		eManualRecipe_SelectedVariableType			: E_XMLVariableType; (* refer to E_XMLVariableType *)
		sManualRecipe_DefaultFilePath				: STRING := 'C:\SW\XML management\Recipe Handling';
		sManualRecipe_FileExtension					: STRING := 'XML';
(**)	sManualRecipe_sErrorMessage					: STRING;
(**)	iManualRecipe_TotalTimePv_100ms				: INT;
(**)	iManualRecipe_ExportedImportedQty			: INT;
(**)	iManualRecipe_ProgressPercentage			: INT;	

(**)	eManualRecipe_ImportExportMode				: E_XmlRWMode; (* refer to E_XmlRwMode :

														eXmlMode_MergeAllByType 					:= 1,			// SSER -> One XML, SSUR -> One XML, Product Recipe -> One XML and so on
														eXmlMode_SeperateByProductAndStation		:= 2,			// SSER will seperate by Station with Multiple file, same goes to the rest of the Recipe
														eXmlMode_SeperateAll					 	:= 3			// Seperate each of the recipe individually *)


	
	eHmiLanguage								: E_HmiLanguage;

	sHmiActiveUsername							: STRING(30):= 'TF2000 HMI User'; 	// Active username that login in HMI currently
	sHmiActiveUsergroup							: STRING(30);
	iHmiCurrentUserIDs							: INT := 1; 						// Standby for HMI Current User used
	ARsHmiUsernameList 							: ARRAY [0..50] OF STRING;			// HMI User Management Namelist push out from HMI
	ARsHmiUsergroupList 						: ARRAY [0..10] OF STRING;			// HMI User Management Namelist push out from HMI
	
	
	bEventRstPB									: BOOL; // Used in program, HMI and any places. This variable need to Mapped with Physical Input via FunctionBlock (FB3_EventModule)
	bBuzzerRstPB								: BOOL; // Used in program, HMI and any places. This variable need to Mapped with Physical Input via FunctionBlock (FB3_EventModule)
	bAcknowledgePB								: BOOL; // Used in program, HMI and any places. This variable need to Mapped with Physical Input via FunctionBlock (FB3_EventModule)
	


// Machine


	bShutdownRequestFlag						: BOOL;
	bManualRecipe_ReadyToShutdownFlag			: BOOL; // 
	bCSVWrite_ReadyToShutdownFlag				: BOOL; // 
	
	
// Boot Up Shut Down
	bMainCtrl									: BOOL;	
	bReadXmlEn									: BOOL;
	bReadXmlComplete							: BOOL;
	bMachineShutdown							: BOOL;
	bShutdownPopupPage							: BOOL;
	bRecipeShutdownRequestFlag					: BOOL;
	bCsvShutdownRequestFlag						: BOOL;
	bWriteXmlEn									: BOOL;
	bWrite_Done									: BOOL;
	bRead_Done									: BOOL;
	
	
// CSV Report Log
		
	dsCsvReport									: DS_CsvReport; // Please consider to change the naming of DS and declaration on upcoming project
	fbBkMemRingBuffer							: FB_MemRingBuffer;
	fbCsvHandler	 							: FB3_CsvHandler;
	sCsvFilePath								: STRING := 'C:\\report_csv\';
	udiCsvMRBCount								: UDINT;	// The number of data set stored in MRB (MemoryRingBuffer)
	udiCsvMRBUsagePercent 						: UDINT;	// Current Usage % in MRB (MemoryRingBuffer)
	ARdsCsvErrorLog								: ARRAY [1..C_iCsvErrorLogQty] OF DS_CsvErrorLog;
	dsCsvErrorLog_Empty							: DS_CsvErrorLog;

// CSV Event Log

	sCsvFilePath_EventLog						: STRING := 'C:\SW\EventLog\';

	
	
END_VAR
	
VAR_GLOBAL PERSISTENT
// Station, Loading, Unloading

//	ARiLdModulePickStnID						: ARRAY [0..C_iLdModuleQty] OF INT;  //XML_AutoRO_ManualRW  	// To "Name" the Loading Station with a Number, usually we will label the 1st Module Loading Conveyor with 79 (7=Loading, 9= the 9th Zone (or we all it max) of the conveyor end zone. 
//	ARiUldModuleUnloadStnID						: ARRAY [0..C_iUldModuleQty] OF INT; //XML_AutoRO_ManualRW		// To "Name" the Unlaoding Station with a Number, usually we will label the 1st Module of Unloading Conveyor with 81 (8=Unloading, 1=The 1st Zone of the unloading Conveyor.
	
// XML Multiple GVL Backup Version

	AR2sXMLMultipleGVLVerDate 				: ARRAY [1..C_iXMLSrvMultiGVLQty] OF ARRAY [1..C_iXMLMultipleGVLVerQty] OF STRING;

(***** CHECK ******


(* xxxxxxxxxxxxxxxxxxxxxxxxxxxxxxx  UPS - Internal Used xxxxxxxxxxxxxxxxxxxxxxxxxxxxxxx*)
(*========================================================================*)

	bGetUpsStatusEn						: BOOL := TRUE;
	bGetUpsStatusValid					: BOOL;
	bGetUpsStatusError					: BOOL;
	udiGetUpsStatusErrID					: UDINT;
	UpsStatus							: ST_UPSStatus;

(* xxxxxxxxxxxxxxxxxxxxxxxxxxxxxxx  UPS - External Used xxxxxxxxxxxxxxxxxxxxxxxxxxxxxxx*)
(*========================================================================*)
	(* --- Alarm --- *)
	bDCPowerUnknownStatusAlarm			: BOOL;
	bBatteryUnknownStatusAlarm			: BOOL;
	bUpsCommUnknownStatusAlarm		: BOOL;
	bBatteryReplacementRequestAlarm		: BOOL;
	bUpsCommErrorAlarm					: BOOL;
	(* --- Status --- *)
	bDCPowerModeActivated				: BOOL;
	bBatteryModeActivated				: BOOL;
	bUpsCommOkFlag					: BOOL;

	timeNow: TIMESTRUCT;

*)
	
(*
	// Arm
	C_iArmModuleQty 				: INT := 1; 								(* Total quantity of Single Arm + Multiple Arm Module - ex: 1x Multiple Arm (with 5 Vertical Axis) + 2x Single Arm = 3 Modules = Value: 3 *)
	C_ARiArmModuleVertAxisQty		: ARRAY [1..C_iArmModuleQty]OF INT := [1];	(* Total quantity of Veritical Axis per Arm Module *)
	C_ARMcArmHookQty				: INT := 1;									(* Total quantity of Hook per Machine, ex: 2x Arm Module, 1st Module with 1x Hook, 2nd Module is Multiple arm with 7x Hook, so thev value is add together = value: 8 *)

	// Station , Loading, Unloading	
	C_iProcessStnQty 						: INT := 6;		(* To change the Qty of Array*)
	C_iLdModuleQty					: INT := 1;		(* To Define Loading Group Set - How many module of Loading Conveyor*)
	C_iUldModuleQty					: INT := 1;		(* To Define Unloading Group Set - How many module of Unloading Conveyor*)
		
	C_ARiCvLdModuleZoneQty			: ARRAY [1..C_iLdStnQty] OF INT := [3];		(* Number of Zone on each of the Loading Conveyor Module (Module seperated by Array) *)
	C_ARiCvUldModuleZoneQty			: ARRAY [1..C_iUldStnQty] OF INT := [3];	(* Number of Zone on each of the Unloading Conveyor Module (Module seperated by Array) *)

	C_iTotalCvLdZoneQty				: INT := 3;		(* Number of Zone on each of the Loading Conveyor Module*)
	C_iTotalCvUldZoneQty			: INT := 3;		(* Number of Zone (Or Max Number of Zone) on each of the Unloading Conveyor Module*)
	*)

	
END_VAR

// ---- GVLs/GVL3/LIB_GVL_IO.TcGVL
{attribute 'Tc2GvlVarNames'}
VAR_GLOBAL


// Digital Input

	ARbDI						: ARRAY [0..C_iDigitalInputQty] OF BOOL;
	ARwMapDI					: ARRAY [100..C_iDigitalInputMappingChannelMaxID] OF WORD;
	ARwActualMapDI	AT %I* 		: ARRAY [1..10] OF WORD;

	
// Digital Output
	ARbDO						: ARRAY [0..C_iDigitalOutputQty] OF BOOL;
	ARwDO						: ARRAY [0..C_iDigitalOutputQty] OF WORD;
	ARwMapDO	 				: ARRAY [100..C_iDigitalOutputMappingChannelMaxID] OF WORD;
	ARwActualMapDO	AT %Q* 		: ARRAY [1..8] OF WORD;
	
// Deactivated

	ARbDeactivated				: ARRAY [0..C_iDigitalOutputQty] OF BOOL;

END_VAR

//VAR_GLOBAL CONSTANT

//	C_iDigitalInputQty					: INT := 220;		// Total Number of Digital Input Points
//	C_iDigitalOutputQty					: INT := 220;		// Total Number of Digital Output Points

//	C_iDigitalInputMappingChannelMaxID	: INT := 150;	// Max Channel ID of Digital Input Channel for Mapping Used (Ex: WX100 ~ WX116 ---> Value: 116
//	C_iDigitalOutputMappingChannelMaxID	: INT := 140; 	// Max Channel ID of Digital Output Channel for Mapping Used (Ex: WY100 ~ WY113 ---> Value: 113
	
//END_VAR

// ---- GVLs/GVL3/LIB_GVL_MEMORY.TcGVL
{attribute 'Tc2GvlVarNames'}
VAR_GLOBAL PERSISTENT
//	AR2dsSSMR						: ARRAY [0..C_iProcessStnQty] OF ARRAY [0..C_iSSMRRecipeQty] OF DS_SSMR;	//XML_AutoRW_ManualRW
//	AR2dsSSUR						: ARRAY [0..C_iProcessStnQty] OF ARRAY [0..C_iSSURRecipeQty] OF DS_SSUR;	//XML_AutoRW_ManualRW
//	AR2dsSSER 						: ARRAY [0..C_iProcessStnQty] OF ARRAY [0..C_iSSERRecipeQty] OF DS_SSER;	//XML_AutoRW_ManualRW
//	ARdsProductRecipe 				: ARRAY [0..C_iProRepRecipeQty] OF DS_ProductRecipe;						//XML_AutoRW_ManualRW

//	dsMcCarrierInfo					: DS_MachineCarrierInfo; 	// Previously call as BasketInfo
//	dsCarrierInfo_Empty				: DS_CarrierInfo;			// Empty DS
	
//	dsSSMR_Empty					: DS_SSMR;
//	dsSSUR_Empty					: DS_SSUR;
//	dsSSER_Empty					: DS_SSER;
//	dsProductRecipe_Empty			: DS_ProductRecipe;
	

	
END_VAR

// ---- GVLs/HMI_Ctrl/Global_Variables_CT12_HMIfunction.TcGVL
{attribute 'Tc2GvlVarNames'}
VAR_GLOBAL

	(*bAutoPageOn:BOOL;
	bManuPageOn:BOOL;
	bRecipePageOn: BOOL;	(*  *)
	bUserPageOn:BOOL;*)


	bSSURstartCOnditionPageOn:BOOL;


	(*bManualStationOnPage:BOOL;*)
	bAutoStationOnPage:BOOL;




END_VAR

// ---- GVLs/HMI_Ctrl/Global_Variables_HMI.TcGVL
{attribute 'Tc2GvlVarNames'}
VAR_GLOBAL

(*Simulator Screen*)

	bSimulatorPagePopUpFlag 							: BOOL;
	bAutoRecipeCallPage 									: BOOL;

	iRecipeSelectNo										: INT;

	bAutoRecipeBarcodeCallPage 							: BOOL;
	bBarcodePagePopUpFlag 								: BOOL;
	bAutoRecipeBarcodeClosePage 						: BOOL;

	sUserName											: STRING;



(*Yoges's Backup and Restore Apps*)

	restore : BOOL;
	backup : BOOL;
	otherwise : BOOL;
	dont : BOOL;
	ask : BOOL;
	me : BOOL;
	silent_backup : BOOL;


	iScrollbar : INT;

END_VAR

// ---- GVLs/HMI_Ctrl/Global_Variables_HMI_Function.TcGVL
{attribute 'Tc2GvlVarNames'}
VAR_GLOBAL PERSISTENT
(*Recipe Setting Page*)

	iStepNo:INT; (*RecipeEditorStepNoAssign*)
	iStationNo:INT;(*BasicRecipeStationNoAssign*)
	iArmStnNo :INT;(*ARm Setting Page*)
	iUsonicID:INT;(*UsonicIDno*)
	iUsonicID2:INT;
	sUltrasonicLabel:STRING;(*UsonicLabel/Name*)
	sUltrasonicLabel2 : STRING;
	iAutoInfoNo:INT;(*AutoMode Station Info Page No*)
	iManuPageNo:INT;(*Manul mode PAge No*)
	iArmControlPageNo:INT; (*Arm Page Control No*)
	OnOffStatus:INT; (*1=System Auto On, 2=System Auto Off*)
	lrVertHmiRatio:LREAL;(*ArmGraphicRatioMovement*)
	lrHorzHmiRatio:LREAL;(*ArmGraphicRatioMovement*)
	bFreqBtmChange: ARRAY [1..iStnQty] OF BOOL;
	bFreqSideChange: ARRAY [1..iStnQty] OF BOOL;	


	(*7day Auto On/Off(array1-On,2=off*)

	Day1En:ARRAY [1..2] OF BOOL;
	Day2En:ARRAY [1..2] OF BOOL;
	Day3En: ARRAY [1..2] OF BOOL;
	Day4En:ARRAY [1..2] OF BOOL;
	Day5En:ARRAY [1..2] OF BOOL;
	Day6En: ARRAY [1..2] OF BOOL;
	Day7En: ARRAY [1..2] OF BOOL;

	Day1H:ARRAY [1..2] OF INT;
	Day2H:ARRAY [1..2] OF INT;
	Day3H: ARRAY [1..2] OF INT;
	Day4H:ARRAY [1..2] OF INT;
	Day5H:ARRAY [1..2] OF INT;
	Day6H: ARRAY [1..2] OF INT;
	Day7H: ARRAY [1..2] OF INT;

	Day1M:ARRAY [1..2] OF INT;
	Day2M:ARRAY [1..2] OF INT;
	Day3M: ARRAY [1..2] OF INT;
	Day4M:ARRAY [1..2] OF INT;
	Day5M:ARRAY [1..2] OF INT;
	Day6M: ARRAY [1..2] OF INT;
	Day7M: ARRAY [1..2] OF INT;

	(*Arm Horizontal Position Remap*)
	Arm1HookPos: ARRAY [0..20] OF LREAL;
	Arm1UnHookPos: ARRAY [0..20] OF LREAL;

	Arm2HookPos: ARRAY [0..20] OF LREAL;
	Arm2UnHookPos: ARRAY [0..20] OF LREAL;

	bAutoPageOn:BOOL;
	bManuPageOn:BOOL;
	bRecipePageOn: BOOL;	(*  *)
	bUserPageOn:BOOL;
	bJRS_PageOn:BOOL;
	bGeneral_PageOn:BOOL;
         bDetergentMonitorAPageOn:BOOL;
         bDetergentMonitorBPageOn:BOOL;
         bVacuumMonitorPageOn:BOOL;
	bManualCalibratePageOn:BOOL;

	xRatio:LREAL;
	yRatio:LREAL;
	xRatio_1:LREAL;
	yRatio_1:LREAL;

	Arm1TopPos: ARRAY [0..iAddMapArrayLreal] OF LREAL;
	Arm1Pos1stStage: ARRAY [0..iAddMapArrayLreal] OF LREAL;
	Arm1Pos2ndStage: ARRAY [0..iAddMapArrayLreal] OF LREAL;
	Arm1Pos3rdStage: ARRAY [0..iAddMapArrayLreal] OF LREAL;
	Arm1Pos4thStage: ARRAY [0..iAddMapArrayLreal] OF LREAL;
	Arm1BottomPos: ARRAY [0..iAddMapArrayLreal] OF LREAL;
	Arm1MidPos: ARRAY [0..iAddMapArrayLreal] OF LREAL;

	Arm2TopPos: ARRAY [0..iAddMapArrayLreal] OF LREAL;
	Arm2Pos1stStage: ARRAY [0..iAddMapArrayLreal] OF LREAL;
	Arm2Pos2ndStage: ARRAY [0..iAddMapArrayLreal] OF LREAL;
	Arm2Pos3rdStage: ARRAY [0..iAddMapArrayLreal] OF LREAL;
	Arm2Pos4thStage: ARRAY [0..iAddMapArrayLreal] OF LREAL;
	Arm2BottomPos: ARRAY [0..iAddMapArrayLreal] OF LREAL;
	Arm2MidPos: ARRAY [0..iAddMapArrayLreal] OF LREAL;

END_VAR

VAR_GLOBAL

	iArmVertCurrentPos:INT;
	iArmHorzCurrentPos:INT;

	bArmPosSetPage:BOOL;
	bArm2PosSetPage : BOOL;


	bDeactivatePageOn:BOOL; (*Sensor Deactivated*)
	bStatusPreparationPageOn:BOOL;

	bArmJog2PageOn: BOOL;

	RecipeEditOn:BOOL; (*RecipeEditorEditPageCallUp*)

	bXML_ImportExportPageOn : BOOL;


	bStatusPreparePageOn:BOOL; (*Open Prepare Status Page*)
	bStatusOriginPageOn:BOOL;	(*Open Origin Status Page*)
	(*bAutoModeOtherDeactPageOn:BOOL;(*Open Deact. Others Page*)*)

	(*Time Tracker & Time Optimize Page*)

	TrackeriArrayNo: ARRAY [1..20] OF INT; (*Assign for tracker Array NO*)
	TimeTrackerPage:INT; (*Assign for tracker Page No*)


	(*Remap Arm Position Function*-because loading/unloading not in array form*)

	(*Produt Description for Recipe Edit*)
	sRecipeDescriptionStep : ARRAY [1..20] OF STRING;

	(*Arm Homing Complete Indicator*)
	bArmVertHomingComplete:BOOL;
	bArmHorzHomingComplete:BOOL;
	bArmHomingComplete: ARRAY [1..iArmQty] OF BOOL;

	(*Page On bit*)

	bAlarmPageOn:BOOL;
	bRecipeSubMenuPageOn:BOOL;

	(*Auto Mode Recipe Select*)
	bAutoModeRecipeSelect:BOOL;

	JogSlowPullOn:BOOL;
	JogArmOn:BOOL;

	(*Station On page bit*)
	bStationOnPage:BOOL;
	bManualStationOnPage:BOOL;
	bManualStationOffPage:BOOL;

	(*Manual Mode U/Sonic Power Set*)

	iUsonicA_PowerManuSV : ARRAY [1..20] OF INT;
	iUsonicB_PowerManuSV : ARRAY [1..20] OF INT;


	(*Detergent Basket Quatity (PV) Reset PB user password control*)
	ARiManualDetergentResetPassword 	: ARRAY [0..iStnQty] OF STRING;
	ARbManualDetergentResetFlag			: ARRAY [0..iStnQty] OF BOOL;

	bInputListOn:BOOL;
	bOutputListOn:BOOL;
	bRecipeListOn:BOOL;


	Xmove:INT;
	Ymove:INT;

	bStationOffPage: BOOL;
	RecipeEditOff:BOOL;
END_VAR

VAR_GLOBAL


END_VAR

// ---- GVLs/Internal Address/GVL_Internal_Variable.TcGVL
{attribute 'Tc2GvlVarNames'}
VAR_GLOBAL
	
	ARbMAP_ArmMisshookSensorA 				: ARRAY [1..iArmQty] OF BOOL;
	ARbMAP_ArmMisshookSensorB 				: ARRAY [1..iArmQty] OF BOOL;
	
	bMAP_LdConfirmBasketPickAvailibility	: BOOL;

END_VAR

// ---- GVLs/Memory_Ctrl/Global_Variables_Memory.TcGVL
{attribute 'Tc2GvlVarNames'}
VAR_GLOBAL PERSISTENT

(* xxxxxxxxxxxsxxxxxx BasketMemory - Basket Cfm/ Trf Internal Used xxxxxxxxsxxxxxxxxx*)
(*========================================================================*)

	fbLdBasketMemory					: ARRAY [0..iCvLdQty] OF fbV2_SingleArmBasketMemoryV2;
	fbA1StationBasketMemory				: ARRAY [0..iStnQty] OF fbV2_SingleArmBasketMemoryV2;
	fbA2StationBasketMemory				: ARRAY [0..iStnQty] OF fbV2_SingleArmBasketMemoryV2;
	fbUldBasketMemory					: ARRAY [0..iCvUldQty] OF fbV2_SingleArmBasketMemoryV2;

(* xxxxxxxxxxxxxxxxxxxxxxxxxxxx  BasketInfo - Internal Used xxxxxxxxxxxxxxxxxxxxxxxxxxxx*)
(*========================================================================*)

	DSLdBasketInfoConfirm 				: ARRAY [0..iLdStnQty] OF DSV2_BasketInfo;
	DSLdBasketInfoTransfer 				: ARRAY [0..iLdStnQty] OF DSV2_BasketInfo;

	DSUldBasketInfoConfirm 				: ARRAY [0..iUldStnQty] OF DSV2_BasketInfo;
	DSUldBasketInfoTransfer 				: ARRAY [0..iUldStnQty] OF DSV2_BasketInfo;

	DSStnBasketInfo						: ARRAY [0..iStnQty] OF DSV2_BasketInfo;
	DSArmBasketInfo 						: ARRAY [0..iArmQty] OF DSV2_BasketInfo;

(* xxxxxxxxxxxxxxxxxxxxx  BasketInfo - Loading / Unloading Conveyor Used xxxxxxxxxxxxxxxxxxxxx *)
(*================================================================================*)

	AR2sDSCv_LdConfirmBasketInfo 		: ARRAY [1..iLdStnQty, 1..iCvLdQty] OF DSV2_BasketInfo;
	AR2sDSCv_LdTransferBasketInfo 		: ARRAY [1..iLdStnQty, 1..iCvLdQty] OF DSV2_BasketInfo;

	AR2sDSCv_UldConfirmBasketInfo 		: ARRAY [1..iUldStnQty, 1..iCvUldQty] OF DSV2_BasketInfo;
	AR2sDSCv_UldTransferBasketInfo 		: ARRAY [1..iUldStnQty, 1..iCvUldQty] OF DSV2_BasketInfo;

(* xxxxxxxxxxxxxxxxxxxxx  Station Memory and InputOutput Variable - Internal Used xxxxxxxxxxxxxxxxxxxxx*)
(*=====================================================================================*)

	LdDSStationSSERStore				: DSV2_fbStationSequenceRecipeStore;
	LdDSStationSSURStore 				: DS_fbStationSubRecipeStore;

	LdDSStationSSERCall					: DSV2_fbStationSequenceRecipeCall;
	LdDSStationSSURCall 					: DS_fbStationSubRecipeCall;

	ARDsStnSeqProInput 					: ARRAY [0..iStnQty] OF DS_StnSeqProInput;
	ARDSStnSeqProOutput 				: ARRAY [0..iStnQty] OF DS_StnSeqProOutput;

	AR10DSStationSSERStore				: ARRAY [0..iStnQty] OF DSV2_fbStationSequenceRecipeStore;
	AR10DSStationSSERCall				: ARRAY [0..iStnQty] OF DSV2_fbStationSequenceRecipeCall;

	AR10DSStationSSURStore 				: ARRAY [0..iStnQty] OF DS_fbStationSubRecipeStore;
	AR10DSStationSSURCall 				: ARRAY [0..iStnQty] OF DS_fbStationSubRecipeCall;

(* xxxxxxxxxxxxxxxxxxxxxxxxxxxxx  Station Process Variable - Internal Used xxxxxxxxxxxxxxxxxxxxxxxxxxxxx*)
(*=====================================================================================*)

	fbMainStationProcess_Stn				: ARRAY [1..iStnQty] OF fbV2_MainStationProcess;
	ARDsStnSeqProcessCtrl 				: ARRAY [0..iStnQty] OF DS_fbStnSeqProcessCtrl;
	ARbProductRecipeCallEn 				: ARRAY [0..iStnQty] OF BOOL;
	ARiProductRecipeNoCall 				: ARRAY [0..iStnQty] OF INT;
	ARiProductRecipeStepCall 				: ARRAY [0..iStnQty] OF INT;
	DSfbGnrProductRecipeMemoryOut 		: DSV2_fbGnrProductRecipeMemoryOut;
	ARiStnNoToCalledArm					: ARRAY [0..iArmQty] OF INT;
	ARDSGnrFeedArmPnpParameter		: ARRAY [0..iArmQty] OF DSV2_Gnr_CalledArmPnpParameter;
	ARbArmReady						: ARRAY [1..iArmQty] OF BOOL;								(* Universal*) (* Input  - From ArmPnpFB, This signal is used to confirm if the arm is ready and idling*)
	ARbStationProcessCompletedFlag		: ARRAY [0..iStnQty] OF BOOL;

(*xxxxxxxxxxxxxxxxxxxxxxxxxxx fbGnrProductRecipeMemory - Internal Used xxxxxxxxxxxxxxxxxxxxxxxxxxx*)
(*=====================================================================================*)

(*Input/Output*)
	ARiCurrentHorzStnNo					: ARRAY [1..iArmQty] OF INT;
	ARi1StepPatternNo					: ARRAY [1..iArmQty] OF INT;
	ARDs1StepUpDownMovement			: ARRAY [1..iArmQty] OF DSA1_UpDownMovement;
	ARi4StepPatternNo					: ARRAY [1..iArmQty] OF INT;
	ARDs4StepUpDownMovement			: ARRAY [1..iArmQty] OF DSA1_UpDownMovement;

(* xxxxxxxxxxxxxxxxxxxxxxxxxxx  Station ZoneHeight Variable - External Used xxxxxxxxxxxxxxxxxxxxxxxxxxx*)
(*=====================================================================================*)

	ARDSLdZoneHeight 					: ARRAY [0..iLdStnQty] OF DSA32_StationZoneHeight;
	ARDSStationZoneHeight 				: ARRAY [0..iStnQty] OF DSA32_StationZoneHeight;
	ARDSUldZoneHeight 					: ARRAY [0..iUldStnQty] OF DSA32_StationZoneHeight;

(* xxxxxxxxxxxxxxxxxxxxxxxxxxx  Station ZoneHeight Variable - Internal Used xxxxxxxxxxxxxxxxxxxxxxxxxxx*)
(*=====================================================================================*)

	ARDSLdZonePosOut					: ARRAY [0..iLdStnQty] OF DSA32_StationZonePosOut; (*From fbGnrProductRecipeMemory Output*)
	ARDSStationZonePosOut 				: ARRAY [0..iStnQty] OF DSA32_StationZonePosOut; (*From fbGnrProductRecipeMemory Output*)
	ARDSUldZonePosOut 					: ARRAY [0..iUldStnQty] OF DSA32_StationZonePosOut;(*From fbGnrProductRecipeMemory Output*)

(* xxxxxxxxxxxxxxxxxxxxxxxxxxxxx  MaxMin Time Used  xxxxxxxxxxxxxxxxxxxxxxxxxxxxx*)
(*====================================================================*)

	ARDsSSERSourceMinMaxTime_Uni		: ARRAY [1..iStnQty] OF DSV2_SSERSourceMinMaxTime;
	ARDsStnMinMaxEffTimeDisplay			: ARRAY [0..iStnQty] OF DSV2_StnMinMaxEffTIme;
	DSV2MTBMinMaxEffTime 				: DSV2_MinMaxEffTime;

(* xxxxxxxxxxxxxxxxxxxxx  IndusoftScreenMapping - External Used xxxxxxxxxxxxxxxxxxxxx*)
(*========================================================================*)

	DSScrMapSSUR 						: DS_fbStationSubRecipeStore;
	DSScrMapSSER 						: DSV2_fbStationSequenceRecipeStore;
	iCurrentScreenNo						: INT;

(* xxxxxxxxxxxxxxxxxxxxx  Indusoft Product Recipe Description Display control  -  xxxxxxxxxxxxxxxxxxxxxxxxxx*)

	ARsUpPickPatternDescription			: ARRAY [0..iProductRecipeStepArrayQty] OF STRING(50);
	ARsDownTransferPatternDescription		: ARRAY [0..iProductRecipeStepArrayQty] OF STRING(50);

(*Indusoft*)
	sProductRecipeStep1SeqRecipeDescription: STRING(50);
	sProductRecipeStep2SeqRecipeDescription: STRING(50);
	sProductRecipeStep3SeqRecipeDescription: STRING(50);
	sProductRecipeStep4SeqRecipeDescription: STRING(50);
	sProductRecipeStep5SeqRecipeDescription: STRING(50);
	sProductRecipeStep6SeqRecipeDescription: STRING(50);
	sProductRecipeStep7SeqRecipeDescription: STRING(50);
	sProductRecipeStep8SeqRecipeDescription: STRING(50);
	sProductRecipeStep9SeqRecipeDescription: STRING(50);
	sProductRecipeStep10SeqRecipeDescription: STRING(50);
	sProductRecipeStep11SeqRecipeDescription: STRING(50);
	sProductRecipeStep12SeqRecipeDescription: STRING(50);
	sProductRecipeStep13SeqRecipeDescription: STRING(50);
	sProductRecipeStep14SeqRecipeDescription: STRING(50);
	sProductRecipeStep15SeqRecipeDescription: STRING(50);
	sProductRecipeStep16SeqRecipeDescription: STRING(50);
	sProductRecipeStep17SeqRecipeDescription: STRING(50);
	sProductRecipeStep18SeqRecipeDescription: STRING(50);
	sProductRecipeStep19SeqRecipeDescription: STRING(50);
	sProductRecipeStep20SeqRecipeDescription: STRING(50);

	ARsUpPickPatternDescription1: STRING(50);
	ARsUpPickPatternDescription2: STRING(50);
	ARsUpPickPatternDescription3: STRING(50);
	ARsUpPickPatternDescription4: STRING(50);
	ARsUpPickPatternDescription5: STRING(50);
	ARsUpPickPatternDescription6: STRING(50);
	ARsUpPickPatternDescription7: STRING(50);
	ARsUpPickPatternDescription8: STRING(50);
	ARsUpPickPatternDescription9: STRING(50);
	ARsUpPickPatternDescription10: STRING(50);
	ARsUpPickPatternDescription11: STRING(50);
	ARsUpPickPatternDescription12: STRING(50);
	ARsUpPickPatternDescription13: STRING(50);
	ARsUpPickPatternDescription14: STRING(50);
	ARsUpPickPatternDescription15: STRING(50);
	ARsUpPickPatternDescription16: STRING(50);
	ARsUpPickPatternDescription17: STRING(50);
	ARsUpPickPatternDescription18: STRING(50);
	ARsUpPickPatternDescription19: STRING(50);
	ARsUpPickPatternDescription20: STRING(50);

	ARsDownTransferPatternDescription1: STRING(50);
	ARsDownTransferPatternDescription2: STRING(50);
	ARsDownTransferPatternDescription3: STRING(50);
	ARsDownTransferPatternDescription4: STRING(50);
	ARsDownTransferPatternDescription5: STRING(50);
	ARsDownTransferPatternDescription6: STRING(50);
	ARsDownTransferPatternDescription7: STRING(50);
	ARsDownTransferPatternDescription8: STRING(50);
	ARsDownTransferPatternDescription9: STRING(50);
	ARsDownTransferPatternDescription10: STRING(50);
	ARsDownTransferPatternDescription11: STRING(50);
	ARsDownTransferPatternDescription12: STRING(50);
	ARsDownTransferPatternDescription13: STRING(50);
	ARsDownTransferPatternDescription14: STRING(50);
	ARsDownTransferPatternDescription15: STRING(50);
	ARsDownTransferPatternDescription16: STRING(50);
	ARsDownTransferPatternDescription17: STRING(50);
	ARsDownTransferPatternDescription18: STRING(50);
	ARsDownTransferPatternDescription19: STRING(50);
	ARsDownTransferPatternDescription20: STRING(50);

END_VAR

// ---- GVLs/ModbusTCP_Ctrl/Global_Variables_Modbus.TcGVL
{attribute 'Tc2GvlVarNames'}
VAR_GLOBAL

(******** Modbus TCP variable declaration - as a SLAVE ********)  (*** If as a MASTER, then don't need to declare this variable***)

   	mb_Input_Coils        		: ARRAY [0..255] OF BOOL;
    	mb_Output_Coils      	 	: ARRAY [0..255] OF BOOL;
    	mb_Input_Registers    		: ARRAY [0..255] OF WORD;
    	mb_Output_Registers   		: ARRAY [0..255] OF WORD;

	bOutputRegisterAddr0		: BOOL;

END_VAR

// ---- GVLs/Others TBD/Globale_VarCheck.TcGVL
{attribute 'Tc2GvlVarNames'}
VAR_GLOBAL
	CheckBounds_ErrCnt:INT;
	CheckByteZeroDiv_ErrCnt:INT;
	CheckDintZeroDiv_ErrCnt:INT;
	CheckDWordZeroDiv_ErrCnt:INT;
	CheckIntZeroDiv_ErrCnt:INT;
	CheckLrealZeroDiv_ErrCnt:INT;
	CheckRealZeroDiv_ErrCnt:INT;
	CheckSIntZeroDiv_ErrCnt:INT;
	CheckWordZeroDiv_ErrCnt:INT;
	CheckRangeSigned_ErrCnt:INT;
	CheckRangeUnsigned:INT;
END_VAR

// ---- GVLs/Others TBD/Global_HMI.TcGVL
{attribute 'Tc2GvlVarNames'}
VAR_GLOBAL

	bAutoModeOnPB		:BOOL;
	bAutoPrepareStatus		:BOOL;
	bBarcodeRegisterPageON	:BOOL;
	bManualModeOnPB	:BOOL;
	bRecipeModeOnPB	:BOOL;
	bRecipeSSUROnPB		:BOOL;
	bRecipeSSEROnPB		:BOOL;
	bRecipeBasicOnPB		:BOOL;
	bRecipeBasic2OnPB		:BOOL;
	bRecipeProductOnPB		:BOOL;
	bRecipeOtherOnPB		:BOOL;
	bRecipeTimeOptimizeOnPB:BOOL;
	bRecipeArmSettingOnPB	:BOOL;
	bRecipeArmSetting2OnPB	:BOOL;
	bAlarmModeOnPB	:BOOL;
	bUserModeOnPB		:BOOL;

	bManualCalibrate		:BOOL;
	bAutoModeOperationStatusPage:	BOOL;


	bAutoModeOn	:BOOL;
	bManualModeOn	:BOOL;
	bRecipeModeOn	:BOOL;
	bRecipeSSUROn	:BOOL;
	bRecipeSSEROn	:BOOL;
	bRecipeBasicOn	:BOOL;
	bRecipeBasic2On	:BOOL;
	bRecipeProductOn:BOOL;
	bRecipeOtherOn	:BOOL;
	bRecipeTimeOptimizeOn:BOOL;
	bRecipeArmSettingOn	:BOOL;
	bRecipeArmSetting2On:BOOL;
	bAlarmModeOn	:BOOL;
	bUserModeOn	:BOOL;
	bSchematicPageOn :BOOL;

	bManualModeOnLatch :BOOL;	(*to call Confirm Pop Up page Manual Out*)
	bManualOutToAutoConfirmPageOn	:BOOL; (*Manual Out Pop Up Page to Auto On bit*)
	bManualOutToRecipeConfirmPageOn	:BOOL; (*Manual Out Pop Up Page to Recipe On bit*)
	bManualOutToUserConfirmPageOn	:BOOL; (*Manual Out Pop Up Page to User On bit*)
	bManualOutLatchCfm				:BOOL; (*Use as a latch bit for timer to reset All Page bit On PB*)
	
	bManualModeOffLatch :BOOL;	(*to exit Confirm Pop Up page Manual Out*)
	bManualOutToAutoConfirmPageOff	:BOOL; (*Manual Out Pop Up Page to Auto Off bit*)
	bManualOutToRecipeConfirmPageOff	:BOOL; (*Manual Out Pop Up Page to Recipe Off bit*)
	bManualOutToUserConfirmPageOff	:BOOL; (*Manual Out Pop Up Page to User Of bit*)




	(*iStationNo		:INT;*)



	bAutoModeOnRE		:R_TRIG;
	bManualModeOnRE	:R_TRIG;
	bRecipeModeOnRE	:R_TRIG;
	bRecipeSSUROnRE	:R_TRIG;
	bRecipeBasicOnRE	:R_TRIG;
	bRecipeBasic2OnRE	:R_TRIG;
	bRecipeSSEROnRE	:R_TRIG;
	bRecipeProductOnRE   :R_TRIG;
	bRecipeOtherOnRE	:R_TRIG;
	bRecipeTimeOptimizeOnRE:R_TRIG;
	bRecipeArmSettingOnRE	:R_TRIG;
	bRecipeArmSetting2OnRE	:R_TRIG;
	bAlarmModeOnRE	:R_TRIG;
	bUserModeOnRE		:R_TRIG;

	bLoadingPageSeqCompleteRE	:R_TRIG;
	bManualModeOnLatchFE	:F_TRIG;


(*Initial Loading Page Timer*)

	bAutoModeOnTON	:TON;
	bManualModeOnTON	:TON;
	bRecipeModeOnTON	:TON;
	bRecipeSSUROnTON	:TON;
	bRecipeSSEROnTON	:TON;
	bRecipeBasicOnTON	:TON;
	bRecipeBasic2OnTON	:TON;
	bRecipeProductOnTON:TON;
	bRecipeOtherOnTON	:TON;
	bRecipeTimeOptimizeOnTON:TON;
	bRecipeArmSettingOnTON	:TON;
	bRecipeArmSetting2OnTON :TON;
	bAlarmModeOnTON	:TON;
	bUserModeOnTON	:TON;
	bManualOutLatchCfmTON 	:TON;


	bAutoModeOnSeq	:BOOL;
	bManualModeOnSeq	:BOOL;
	bRecipeModeOnSeq	:BOOL;
	bRecipeSSUROnSeq	:BOOL;
	bRecipeSSEROnSeq	:BOOL;
	bAlarmModeOnSeq	:BOOL;
	bUserModeOnSeq	:BOOL;
         bRecipeBasicOnSeq	:BOOL;
         bRecipeBasic2OnSeq	:BOOL;
         bRecipeProductOnSeq		:BOOL;
	bRecipeOtherOnSeq		:BOOL;
	bRecipeTimeOptimizeOnSeq:BOOL;
	bRecipeArmSettingOnSeq	:BOOL;
	bRecipeArmSetting2OnSeq	:BOOL;


(*Password Save Confirm page*)
	bSaveCfmPB: BOOL;
	bSaveCfmPageOn: BOOL;
	bSaveBufferPB:BOOL;
	bSavePageCnfmOnRE: R_TRIG;
	sUserPasswordSave: STRING;
	tBackupDelayOffTimer: TON;
	bIncorrectPswdOn: BOOL;
	bSaveBufferPBRE: R_TRIG;



(*Xml Execute Push Button*)
	bExecuteWriteXml		: BOOL;
	bExecuteReadXml	:BOOL;
	bErrorReadXml		:BOOL;


(*Secs\Gem Command Page Call*)

	bSecGemsPageON 									:BOOL;

(*Recipe Selection Mode*)

	sRecipeSelectionStatus								:STRING;

(*SECS\GEM Selection Mode Message*)

	sSecGemSelectionButtonMessage						:STRING;

	sRemotCommandStateMessage						:STRING;





	bLoadingPageSeqComplete	:BOOL;
	
	ARdsMAP_HmiVariableStn		: ARRAY[1..iStnQty] OF DS_HMI_MappingVariable;
	ARdsMAP_HmiVariableGeneral	: DS_HMI_MappingVariable;

	
END_VAR

// ---- GVLs/Others TBD/Global_Variables_Lib_NonPresistent.TcGVL
{attribute 'Tc2GvlVarNames'}
VAR_GLOBAL

(*Global Variable for FunctionBlock in Library *)

	(* HMI Declaration *)
	iHMIRecipeNo				: INT;
	bRecipeLoadPb				: BOOL;
	bRecipeSavePb				: BOOL;
	bProductRecipeClearPb		: BOOL;
	bClearPB_SSER 				: ARRAY [1..6] OF BOOL;
	bClearPB_SSUR 				: ARRAY [1..6] OF BOOL;
	bClearPB_SSER_Uni			: BOOL;
	bClearPB_SSUR_Uni			: BOOL;
	

	(*XML Handler & XML Fb*)
	iXMLRecipeNo				: INT := 1;
	FBXmlSrvRead				:  FB_XmlSrvRead;
	FBXmlSrvWrite				:  FB_XmlSrvWrite;
	DSV3XML_Recipe			: DSV3_XML_Recipe;

	ARiSubAction					: ARRAY [1..10] OF INT; (* 0-Idle, 1-Import, 2-Export, 3-Clear/Delete 8-Done *)



	(*SecsGem Simulation Used Only*)

	iSecsGemRecipeNo			: INT := 1;

	iSecsGemLoadHS			: INT; 				(* S7F1/S7F2 		: 0-Idle, 1-Enable, 2-Busy, 3-Done, 4-Error *)
	iSecsGemSentHS				: INT; 				(* S7F3/S7F4 		: 0-Idle, 1-Enable, 2-Busy, 3-Done, 4-Error *)
	iSecsGemRequestHS			: INT; 				(* S7F5/S7F6 		: 0-Idle, 1-Enable, 2-Busy, 3-Done, 4-Error *)
	iSecsGemDeleteHS			: INT; 				(* S7F17/S7F18 	: 0-Idle, 1-Enable, 2-Busy, 3-Done, 4-Error *)


	(* Declared for S7F18 -> Delete Request *)
	ARDsPnpSequenceMemory_Delete 									: ARRAY [1..iProductRecipeArrayQty] OF DSV2_A1_PnpSequenceMemory;
	AR3SiRecipeTimeBlockMemoryNoCallArmTime_Delete				    : ARRAY [1..iProductRecipeArrayQty, 1..iRecipeBlockQty, 1..9] OF INT;
	AR3SiRecipeTimeBlockMemoryWithCallArmTime_Delete				: ARRAY [1..iProductRecipeArrayQty, 1..iRecipeBlockQty, 1..9] OF INT;
	ARbProductRecipeTimeBlockAvailable_Delete 						: ARRAY [0..iProductRecipeArrayQty] OF BOOL;
	ARDSTempCtrlRecipe_Delete 										: ARRAY [0..iProductRecipeArrayQty] OF DSV3_TempCtrlRecipe;


END_VAR

// ---- GVLs/Others TBD/Global_Variables_Lib_Persistent.TcGVL
{attribute 'Tc2GvlVarNames'}
VAR_GLOBAL PERSISTENT


	ARiLdStnID								: ARRAY [1..iLdStnQty] OF INT;		(* To Define Loading Station ID*)
	ARiUldStnID								: ARRAY [1..iUldStnQty] OF INT;		(* To Define Unloading Station ID*)

	ARDSTempCtrlRecipe 					: ARRAY [0..iProductRecipeArrayQty] OF DSV3_TempCtrlRecipe;  (* Used by fbV3_TemperatureParaRecipe, Make it Global so that future can read/write easily*)

END_VAR

// ---- GVLs/Others TBD/Global_Variables_PID.TcGVL
{attribute 'Tc2GvlVarNames'}
VAR_GLOBAL

	No_input							: INT;
	Ratio								: INT;
	InvRatio							: INT;

	Stn1FlowRawData				: INT;
	Stn2FlowRawData				: INT;
	Stn3FlowRawData				: INT;
	Stn4FlowRawData				: INT;
	Stn5FlowRawData				: INT;
	Stn6FlowRawData				: INT;
	Stn7FlowRawData				: INT;
	ARiStnFlowRawData				: ARRAY [1..iStnQty] OF INT;

	Stn1ActualFlowRawData		: INT;
	Stn2ActualFlowRawData		: INT;
	Stn3ActualFlowRawData		: INT;
	Stn4ActualFlowRawData		: INT;
	Stn5ActualFlowRawData		: INT;
	Stn6ActualFlowRawData		: INT;
	Stn7ActualFlowRawData		: INT;
	ARiStnActualFlowRawData	: ARRAY [1..iStnQty] OF INT;


	Stn1U_SonicOn				: BOOL;
	Stn2U_SonicOn				: BOOL;
	Stn3U_SonicOn				: BOOL;
	Stn4U_SonicOn				: BOOL;
	Stn5U_SonicOn				: BOOL;
	Stn6U_SonicOn				: BOOL;
	Stn7U_SonicOn				: BOOL;
	ARiStnU_SonicOn			: ARRAY [1..iStnQty] OF BOOL;

	Pump1_Freq_Reading			: REAL;
	Pump2_Freq_Reading			: REAL;
	Pump3_Freq_Reading			: REAL;
	Pump4_Freq_Reading			: REAL;
	Pump5_Freq_Reading			: REAL;
	Pump6_Freq_Reading			: REAL;
	Pump7_Freq_Reading			: REAL;

	Pump1_Freq_Actual			: INT;
	Pump2_Freq_Actual			: INT;
	Pump3_Freq_Actual			: INT;
	Pump4_Freq_Actual			: INT;
	Pump5_Freq_Actual			: INT;
	Pump6_Freq_Actual			: INT;
	Pump7_Freq_Actual			: INT;

	Pump1_Freq_Reading_Raw	: INT;
	Pump2_Freq_Reading_Raw	: INT;
	Pump3_Freq_Reading_Raw	: INT;
	Pump4_Freq_Reading_Raw	: INT;
	Pump5_Freq_Reading_Raw	: INT;
	Pump6_Freq_Reading_Raw	: INT;
	Pump7_Freq_Reading_Raw	: INT;

	Stn1Actual_LPM				: INT;
	Stn2Actual_LPM				: INT;
	Stn3Actual_LPM				: INT;
	Stn4Actual_LPM				: INT;
	Stn5Actual_LPM				: INT;
	Stn6Actual_LPM				: INT;
	Stn7Actual_LPM				: INT;

	Pump1FlowAlarm				: BOOL;
	Pump2FlowAlarm				: BOOL;
	Pump3FlowAlarm				: BOOL;
	Pump4FlowAlarm				: BOOL;
	Pump5FlowAlarm				: BOOL;
	Pump6FlowAlarm				: BOOL;
	Pump7FlowAlarm				: BOOL;
	
	//Heater
	Stn8TempRawData				: INT;
	Stn9TempRawData				: INT;
	Stn10TempRawData			: INT;



END_VAR

// ---- GVLs/Others TBD/Global_Variables_PID_1.TcGVL
{attribute 'Tc2GvlVarNames'}
VAR_GLOBAL PERSISTENT


	Stn1PumpHiFlowSV		:INT;
	Stn2PumpHiFlowSV		:INT;
	Stn3PumpHiFlowSV		:INT;
	Stn4PumpHiFlowSV		:INT;
	Stn5PumpHiFlowSV		:INT;
	Stn6PumpHiFlowSV		:INT;
	Stn7PumpHiFlowSV		:INT;
	ARiStnPumpHiFlowSV	:ARRAY [1..iStnQty] OF INT;


	Stn1PumpLowFlowSV	:INT;
	Stn2PumpLowFlowSV	:INT;
	Stn3PumpLowFlowSV	:INT;
	Stn4PumpLowFlowSV	:INT;
	Stn5PumpLowFlowSV	:INT;
	Stn6PumpLowFlowSV	:INT;
	Stn7PumpLowFlowSV	:INT;
	ARiStnPumpLowFlowSV	: ARRAY [1..iStnQty] OF INT;

	ARiStnManualPumpLowFlowSV :ARRAY [1..iStnQty] OF INT;
	ARiStnManualPumpHighFlowSV :ARRAY [1..iStnQty] OF INT;


END_VAR

// ---- GVLs/Others TBD/GVL_HMI_CKK.TcGVL
{attribute 'Tc2GvlVarNames'}
VAR_GLOBAL


	
	iBufferPage											: INT;
	iSelectedPage										: INT;
	iReturnPage											: INT;
	bManualPageOn										: BOOL;
	bManualExitConfirm									: BOOL;
	bManualExitCancel									: BOOL;
	bBlockBasketEnter									: BOOL;
iCkkTest	: DINT;


iDisplayTimeCycle : ARRAY [1..iStnQty] OF REAL; 
bDisplayTimeCycleOn : ARRAY [1..iStnQty] OF BOOL;
iDisplayTimeCycleEnd : ARRAY [1..iStnQty] OF INT;
ARiStnProcessTimeCD : ARRAY [1..iStnQty] OF INT;
ARsStnProcessName : ARRAY [1..iStnQty] OF STRING;
iAutoStnInfoPageNo	: INT :=1;
ARsHMIDisplaySSURDescription	: ARRAY [1..IStationSubRecipeArrayQty] OF STRING;
iSettingStnNo	: INT :=1;
iSettingStnNoBuffer	: INT :=1;
iArmSettingStnNo : INT :=1;
iArmSettingStnNoBuffer : INT :=1;
sDisplayConductivity : ARRAY [1..2] OF STRING;
bDosingPageEn		 : ARRAY [1..iStnQty] OF BOOL;
iConfigSSER			 : ARRAY [1..20] OF INT;
bSelectTempExternal	 : ARRAY [1..4] OF BOOL;
bSelectTempExternalInd : ARRAY [1..4] OF BOOL;
iSelectTempExternal	 : INT;
bBarcodeRegPage		 : BOOL;
iDisplayFreqUs		 : ARRAY [1..iStnQty] OF INT;
iDisplayRecipeFreqUs : INT;

sBasketNo			 : STRING;
bBarcodeConfirm		 : BOOL;

bParameterPopupPageOn : BOOL;

bPopupPageRapidPBOn: BOOL;
bPopupPageRapidConfirm: BOOL;
bBarcodeCallPagePB		: BOOL;

// Barcode
sBarcodeScannerReceivedResult: STRING;
	iBarcodeRegUserSelectRecipeNo			: INT;
	iBarcodeRegUserSelectNoDataToSave		: INT;
	bBarcodeRegSave							: BOOL;
	bBarcodeRegClear						: BOOL;
	//bBarcodeEmpty							: BOOL;
	
	bBufferClearPB_SSER 				: ARRAY [1..6] OF BOOL;
	bBufferClearPB_SSUR 				: ARRAY [1..6] OF BOOL;
	
	tClearPB_SSER_Timer 				: ARRAY [1..6] OF TON;
	tClearPB_SSUR_Timer 				: ARRAY [1..6] OF TON;
	
	
END_VAR

// ---- GVLs/PDF_Report/Global_Variables_PDF_Report.TcGVL
{attribute 'Tc2GvlVarNames'}
VAR_GLOBAL

	sNameUser	:STRING;													(*Map with User login Name*)

	a1_dataLink								: ARRAY [1..100] OF ST_DataLog;
	a2_dataLink								: ARRAY [1..100] OF ST_DataLog;
	a3_dataLink								: ARRAY [1..100] OF ST_DataLog;
	a4_dataLink								: ARRAY [1..100] OF ST_DataLog;
	a5_dataLink								: ARRAY [1..100] OF ST_DataLog;
	a6_dataLink								: ARRAY [1..100] OF ST_DataLog;
	a7_dataLink								: ARRAY [1..100] OF ST_DataLog;
	a8_dataLink								: ARRAY [1..100] OF ST_DataLog;
	a9_dataLink								: ARRAY [1..100] OF ST_DataLog;
	a10_dataLink								: ARRAY [1..100] OF ST_DataLog;
	a11_dataLink								: ARRAY [1..100] OF ST_DataLog;
	a12_dataLink								: ARRAY [1..100] OF ST_DataLog;

	sLdtittle								: STRING;
	sStn1tittle								: STRING;
	sStn2tittle								: STRING;
	sStn3tittle								: STRING;
	sStn4tittle								: STRING;
	sStn5tittle								: STRING;
	sStn6tittle								: STRING;
	sStn7tittle								: STRING;
	sStn8tittle								: STRING;
	sStn9tittle								: STRING;
	sStn10tittle								: STRING;
	sStn11tittle								: STRING;
	sStn12tittle								: STRING;
	sStn13tittle								: STRING;

	
	ARsLdBasketInTime 					: ARRAY [0..iLdStnQty] OF STRING;
	ARsStnBasketInTime 					: ARRAY [0..iStnQty] OF STRING;
	ARsStnBasketOutTime 				: ARRAY [0..iStnQty] OF STRING;
	ARsUldBasketInTime 					: ARRAY [0..iUldStnQty] OF STRING;
	
	ARiLdBasketProductRecipeBuffer 		: ARRAY [0..iLdStnQty] OF INT;
	ARsLdBasketNoBuffer 				: ARRAY [0..iLdStnQty] OF STRING;
	
	ARiStnBasketProductRecipeBuffer 	: ARRAY [0..iStnQty] OF INT;
	ARsStnBasketNoBuffer 				: ARRAY [0..iStnQty] OF STRING;
	
	ARiUldBasketProductRecipeBuffer 	: ARRAY [0..iUldStnQty] OF INT;
	ARsUldBasketNoBuffer 				: ARRAY [0..iUldStnQty] OF STRING;
	
END_VAR

VAR_GLOBAL PERSISTENT

	iProgBatchTotal							:INT; (*For Unique nobor for each file*)

END_VAR

// ---- GVLs/Process_Ctrl/Global_Variables_Process_NoPersistent.TcGVL
{attribute 'Tc2GvlVarNames'}
VAR_GLOBAL

(* xxxxxxxxxxxxxxxxxxxxxxx DosingPumpControl Process Variable xxxxxxxxxxxxxxxxxxxxxxx*)
(*========================================================================*)

(*Input*)
	ARbStnErrorReset										: ARRAY [1..iStnQty] OF BOOL;
	ARbStnDrainST										: ARRAY [1..iStnQty] OF BOOL;
	ARbStnManualDosingST 								: ARRAY [1..iStnQty] OF BOOL;
	ARbStnFirstFillST										: ARRAY [1..iStnQty] OF BOOL;
	ARbStnAutoDosingST									: ARRAY [1..iStnQty] OF BOOL;

(*Output*)

	ARbStnAutoDosingDone 								: ARRAY [1..iStnQty] OF BOOL;
	ARbStnManualDosingDone 							: ARRAY [1..iStnQty] OF BOOL;
	ARbStnFirstFillInProgress 								: ARRAY [1..iStnQty] OF BOOL;
	ARbStnAutoDosingInProgress 							: ARRAY [1..iStnQty] OF BOOL;
	ARbStnManualDosingInProgress 						: ARRAY [1..iStnQty] OF BOOL;
	ARbStnPumpHealthCheckPulseError						: ARRAY [1..iStnQty] OF BOOL;

	ARiStnHealthCheckPulsePV							: ARRAY [1..iStnQty] OF INT;

	ARbStnFirstFillingHR									: ARRAY [1..iStnQty] OF BOOL;
	ARbStnFirstFillDone									: ARRAY [1..iStnQty] OF BOOL;

(* xxxxxxxxxxxxxxxxxxxxxxxxxxxxx Conveyor Motor Control xxxxxxxxxxxxxxxxxxxxxxxxxxxxx*)
(*========================================================================*)

	ARbLdIndexPB 										: ARRAY [0..iLdStnQty] OF BOOL;
	ARsLdConvStatus										: ARRAY [0..iLdStnQty] OF STRING;

	ARbUldIndexPB 										: ARRAY [0..iUldStnQty] OF BOOL;
	ARsUldConvStatus									: ARRAY [0..iUldStnQty] OF STRING;

	ARbLdConveyorIdErrorFlag 							: ARRAY [1..iCvLdQty] OF BOOL;
	ARbUldConveyorIdErrorFlag 							: ARRAY [1..iCvUldQty] OF BOOL;

	ARtLdIndexPBDelayTimePV 							: ARRAY [0..iLdStnQty] OF TIME;
	ARtLdRapidPBDelayTimePV 							: ARRAY [0..iLdStnQty] OF TIME;
	ARtLdTimerBasedRapidDelayTimePV					: ARRAY [0..iLdStnQty] OF TIME;
	ARtLdIndexConfirmDelayTimePV 						: ARRAY [0..iLdStnQty] OF TIME;
	ARtLdEndZoneDelayTimePV 							: ARRAY [0..iLdStnQty] OF TIME;

	ARtUldIndexPBDelayTimePV 							: ARRAY [0..iUldStnQty] OF TIME;
	ARtUldRapidPBDelayTimePV 							: ARRAY [0..iUldStnQty] OF TIME;
	ARtUldTimerBasedRapidDelayTimePV					: ARRAY [0..iUldStnQty] OF TIME;
	ARtUldIndexConfirmDelayTimePV 						: ARRAY [0..iUldStnQty] OF TIME;
	ARtUldEndZoneDelayTimePV 							: ARRAY [0..iUldStnQty] OF TIME;

	bConveyorStartInternal									: BOOL;
	bConveyorInternal											: BOOL	;

	Ld1ConvFb											: fbV2_LdUldCvCtrl;
	Uld1ConvFb											: fbV2_LdUldCvCtrl;
	Uld2ConvFb											: fbV2_LdUldCvCtrl;

	fbV2LdCv5zonewith5m5sCtrl								: fbV2_Cv5zonewith5m5sCtrl;
	fbV2LdCv4zonewith4m4sCtrl								: fbV2_Cv4zonewith4m4sCtrl;
	fbV2LdCv3zonewith3m3sCtrl								: fbV2_Cv3zonewith3m3sCtrl;
	bLdCvBasketEndReached								: BOOL;
	bLdCvBasketFull										: BOOL;

	fbV2UldCv5zonewith5m5sCtrl							: fbV2_Cv5zonewith5m5sCtrl;
	fbV2UldCv4zonewith4m4sCtrl							: fbV2_Cv4zonewith4m4sCtrl;
	fbV2UldCv3zonewith3m3sCtrl							: fbV2_Cv3zonewith3m3sCtrl;
	bUldCvBasketEndReached								: BOOL;
	bUldCvBasketFull										: BOOL;

(* xxxxxxxxxxxxxxxxxxxxxxxxxxxxx AutoPreparation Variable xxxxxxxxxxxxxxxxxxxxxxxxxxxxx*)
(*========================================================================*)

	ARtStnDelayOffTopupTimerOn							: ARRAY [0..iStnQty] OF TON;
	ARtStnSubTankDelayOffTopupTimerOn					: ARRAY [0..iStnQty] OF TON;
	ARtMainTankDelayOffTopupTimerOn						: TON;
	ARtMainTankRowDelayOffTopupTimerOn					: TON;
	ARtLoadingRowDelayOffTopupTimerOn					: TON;

	ARtStnTimeEV										: ARRAY [0..iStnQty] OF TIME;
	ARtStnSubTankTimeEV								: ARRAY [0..iStnQty] OF TIME;
(* xxxxxxxxxxxxxxxxxxxxxxxxxx Manual Drain Process Variable xxxxxxxxxxxxxxxxxxxxxxxxxx*)
(*========================================================================*)

	ARtStnDrainLowLevelDelayTimer						: ARRAY [0..iStnQty] OF TON;

	ARtStnDrainDelayEV									: ARRAY [0..iStnQty] OF TIME;

	bManualAllTankDrainEn 								: BOOL;
	bManualAllTankDrainCompletedFlag						: BOOL;

(* xxxxxxxxxxxxxxxxxxxxxxxxxx  Process Variable xxxxxxxxxxxxxxxxxxxxxxxxxx*)
(*========================================================================*)

	ARbStnCylinderInOutCtrl 								: ARRAY [1..iStnQty] OF BOOL;
	ARbStnCylinderOriginFlag								: ARRAY [1..iStnQty] OF BOOL;

(* xxxxxxxxxxxxxxxxxxxxxxxxxxx Vacuum Drain Variable Cltr xxxxxxxxxxxxxxxxxxxxxxxxxxx*)
(*========================================================================*)

	bCCtankDrainDone									: BOOL;
	bManualClearWaterTrap								: BOOL;
	bStnManualDrainCut									: BOOL;

(* xxxxxxxxxxxxxxxxxxxxxxxxxxxxxxxx General Process Variable xxxxxxxxxxxxxxxxxxxxxxxxxxxxxxxx*)
(*========================================================================*)

	ARiStnToleranceTimePV								: ARRAY [0..iStnQty] OF INT;
	ARbStnAssignBadBskBit								: ARRAY [0..iStnQty] OF BOOL;
	bBasketMissingReset									: BOOL;


(* xxxxxxxxxxxxxxxxxxxxxxxxxxxxxxxx Station Min  Process Time Displayed Variable xxxxxxxxxxxxxxxxxxxxxxxxxxxxxxxx*)
(*========================================================================*)
	fbV3TotalProcessTimeTracker							: fbV3_TotalProcessTimeTracker;
	ARiStationMinTimeDisplay								: ARRAY [1..iStnQty] OF INT;
	sStationDescriptionDisplay								: STRING;



END_VAR

// ---- GVLs/Process_Ctrl/Global_Variables_Process_Persistent.TcGVL
{attribute 'Tc2GvlVarNames'}
VAR_GLOBAL PERSISTENT

(* xxxxxxxxxxxxxxxxxxxxxxx DosingPumpControl Process Variable xxxxxxxxxxxxxxxxxxxxxxx*)
(*========================================================================*)

	ARDSProminentDosingHMI 									: ARRAY [1..iStnQty] OF DS_ProminentDosingHMI;
	ARfbProminentDosingCtrl									: ARRAY [1..iStnQty] OF fbProminentDosingCtrl;

	ARiStnPulseOnTime_ms									: ARRAY [1..iStnQty] OF INT;
	ARiStnPulseOffTime_ms 									: ARRAY [1..iStnQty] OF INT;
	ARiStnPumpFeedbackPulseInputFilter_ms 					: ARRAY [1..iStnQty] OF INT;
	ARiStnPumpHealthCheckPulseSV 							: ARRAY [1..iStnQty] OF INT;

(* xxxxxxxxxxxxxxxxxxxxxxxxxxxxx Conveyor Motor Control xxxxxxxxxxxxxxxxxxxxxxxxxxxxx*)
(*========================================================================*)

	ARrLdIndexPBDelayTimeSV_Sec 							: ARRAY [0..iLdStnQty] OF REAL;
	ARrLdRapidPBDelayTimeSV_Sec 							: ARRAY [0..iLdStnQty] OF REAL;
	ARrLdIndexConfirmDelayTimeSV_Sec 						: ARRAY [0..iLdStnQty] OF REAL;
	ARrLdEndZoneDelayTimeSV_Sec 							: ARRAY [0..iLdStnQty] OF REAL;

	ARrUldIndexPBDelayTimeSV_Sec 							: ARRAY [0..iUldStnQty] OF REAL;
	ARrUldRapidPBDelayTimeSV_Sec 							: ARRAY [0..iUldStnQty] OF REAL;
	ARrUldIndexConfirmDelayTimeSV_Sec 						: ARRAY [0..iUldStnQty] OF REAL;
	ARrUldEndZoneDelayTimeSV_Sec 							: ARRAY [0..iUldStnQty] OF REAL;

	diUnloadingTimer										: DINT;
	diUnloadingSingleBasketReachedTimer						: DINT;
	diUnloadingBuzzerOffHeaterTimer							: DINT;
	iUldBasketDelayPushTimerSV_sec							: INT;
	iUldBasketDelayPushTimeCountDown						: INT;
	diLdReturnConvMotorDelayOffTimer						: DINT;
	diUldReturnConvMotorDelayOffTimer						: DINT;

	rLdConveyorPos1ConfirmDelayTimeSV_Sec 					: REAL;
	rLdConveyorPos2ConfirmDelayTimeSV_Sec 					: REAL;
	rLdConveyorPos3ConfirmDelayTimeSV_Sec 					: REAL;
	rLdConveyorPos4ConfirmDelayTimeSV_Sec 					: REAL;

	rLdConveyorPos1ConfirmDelayOnTimeSV_Sec 				: REAL;
	rLdConveyorPos2ConfirmDelayOnTimeSV_Sec 				: REAL;
	rLdConveyorPos3ConfirmDelayOnTimeSV_Sec 				: REAL;
	rLdConveyorPos4ConfirmDelayOnTimeSV_Sec 				: REAL;
	
	rUldConveyorPos1ConfirmDelayTimeSV_Sec 					: REAL;
	rUldConveyorPos2ConfirmDelayTimeSV_Sec 					: REAL;
	rUldConveyorPos3ConfirmDelayTimeSV_Sec 					: REAL;
	rUldConveyorPos4ConfirmDelayTimeSV_Sec 					: REAL;

	rUldConveyorPos1ConfirmDelayOnTimeSV_Sec 				: REAL;
	rUldConveyorPos2ConfirmDelayOnTimeSV_Sec 				: REAL;
	rUldConveyorPos3ConfirmDelayOnTimeSV_Sec 				: REAL;
	rUldConveyorPos4ConfirmDelayOnTimeSV_Sec 				: REAL;

(* xxxxxxxxxxxxxxxxxxxxxxxxxxx General Process Variable xxxxxxxxxxxxxxxxxxxxxxxxxxx*)
(*======================================================================*)

	ARiStnToleranceTimeSV									: ARRAY [0..iStnQty] OF INT;
	ARiArmToleranceTimeSV									: ARRAY [0..iArmQty] OF INT;

	ARbRecipeSelectedFlag									: ARRAY [1..iProductRecipeArrayQty] OF BOOL;

         ARbOptionSelectedAutoTopupFlag						          : ARRAY [1..iProductRecipeArrayQty] OF BOOL;
         ARbOptionSelectedRecipeFlag						      	  	 : ARRAY [1..iProductRecipeArrayQty] OF BOOL;

(* xxxxxxxxxxxxxxxxxxxxxxxxxxx Arm related in Process xxxxxxxxxxxxxxxxxxxxxxxxxxx*)
(*======================================================================*)

	tAllStnArmTake											: INT;
	ARiStnDippingTimeSV										: ARRAY [1..iStnQty] OF INT;
	iFFUDelayOffTimerSV_min									: INT;
	iStnAgitation1DelayOffTimerSV_min							: INT;
	iStnAgitation2DelayOffTimerSV_min							: INT;

(* xxxxxxxxxxxxxxxxxxxxxxxxxxxxx Valve related in Process  xxxxxxxxxxxxxxxxxxxxxxxxxxxxx*)

	iAllTankLowLevelDelayTimeSV 							: INT;
	ARiLoadingTopUpDelayOffTimeSV 							: INT;
	ARiStnTopUpDelayOffTimeSV								: ARRAY [1..iStnQty] OF INT;
	ARiStnSubTankTopUpDelayOffTimeSV						: ARRAY [1..iStnQty] OF INT;

	ARiStnTopUpMaxTimeCutOffSV								: ARRAY [1..iStnQty] OF INT;

	iVacuumDrainSV											: INT;

	bBasketPushBasedTimer									: BOOL;

	ARbIncomingDIValveBasedDetergent						: ARRAY [1..iStnQty] OF BOOL;

	iCylinderBasketBackDelayTimeSV							: INT;
	iCylinderBasketFrontDelayTimeSV							: INT;

	iStn3PumpHzSV												: INT;

(* xxxxxxxxxxxxxxxxxxxxxxxxxxxxxxxx Dryer Cooling Ctrl xxxxxxxxxxxxxxxxxxxxxxxxxxxxxxxx*)
(*========================================================================*)

	ARfbV2DryerCoolingCtrlStn 									: ARRAY [1..iStnQty] OF fbV2_DryerCoolingCtrl;
	ARsStnDryerCoolingStatus									: ARRAY [1..iStnQty] OF STRING;
	ARiStnHeaterOnTimeActivation_Sec 							: ARRAY [1..iStnQty] OF INT ;
	ARiStnBlowerDelayOffTime_min								: ARRAY [1..iStnQty] OF INT ;

END_VAR

// ---- GVLs/RecycleMachineJRSCtrl/Global_Variables_JRS_HMI.TcGVL
{attribute 'Tc2GvlVarNames'}
VAR_GLOBAL

(*JRS_HMI Function*)

	JrsHmiPage:INT;
	bChillerManualPageOn:BOOL;
	bChillerAutoPageOn:BOOL;
	bManulBoilPageOn:BOOL;


END_VAR

// ---- GVLs/RecycleMachineJRSCtrl/Global_Variables_RecycleJRS.TcGVL
{attribute 'Tc2GvlVarNames'}
VAR_GLOBAL PERSISTENT

	DSV3_JRSHMI 											: DSV3_JRS_HMI; (*Channel of Other Digitial IO and DT*)

END_VAR

VAR_GLOBAL

	fbV3JRSModuleWithChiller									: fb_V3JRSModuleWithChiller;

	DSV3_JRSAlarm 											: DSV3_JRS_Alarm; (*Channel 200 ~ 204*)
	DSV3_JRSInput 											: DSV3_JRS_Input; (*Channel 0 ~ 3 *)
	DSV3_JRSOutput 											: DSV3_JRS_Output; (*Channel 100 ~ 103*)


END_VAR

// ---- GVLs/Secs_Gem/Global_Secs_Gem.TcGVL
{attribute 'Tc2GvlVarNames'}
VAR_GLOBAL

(*Machine Status & Control*)
(*-----------------------------------------------------------------------------------------------------------------------------------------------------------------------------------------------------------------------------------------------------------------*)

	(*Remote Command*)
	iRemote_Command_State : INT; (*Command from Secs/Gem to remote machine (Function only in Online Remote)
								 0 - Idle, 1 - INIT, 2 - RESET, 3 - START, 4 - STOP, 5 - PP-SELECT*)

	(*(*Control State-In Persisten Page*)
	iSecs_Control_State :INT;	(* Determine in Gem Console. Machine react base on this setting
							3 - Offline (Secs/GEM Offline - Remote Command disable)
							4 - Online Local (Secs/GEM Online - Local Control - Remote Command disable)
							5 - Online Remote (Secs/Gem Online - Host Control - Remote Command enable)*)*)

	(*Machine Status/ Process Status*)
	iMachine_Status :INT; 		(*Update Secs/Gem the Machine Status
							1 - INIT, 2 - READY, 3 - RUNNING, 4 - ALARM, 5 - STOP*)

	iSecGemStationNo	:INT; (*To refresh the station no for data (Constant Variable*)
(*Control State*)



(*-----------------------------------------------------------------------------------------------------------------------------------------------------------------------------------------------------------------------------------------------------------------*)



(*Production Info /Basket Info*)
(*-----------------------------------------------------------------------------------------------------------------------------------------------------------------------------------------------------------------------------------------------------------------*)

	(*Input Basket ID*)
	(*AR2sDSCv_LdConfirmBasketInfo[1,1].sProgramDescription		:STRING; (*Update Secs/Gem the Basket In ID UPH - Secs/Gem able to capture the start process
																	  (Update Sequence - PPExecName -> Input Basket ID)*)
	(*Output Basket ID*)
	AR2sDSCv_UldConfirmBasketInfo[1,3].sProgramDescription		:STRING;  (*Update Secs/Gem the Basket Out ID, Result & Counter UPH - Secs/Gem able to capture the end process
																	   (Update Sequence - Output Basket Result -> Output Basket Counter -> Output Basket ID)*)
	(*Output Basket Result*)
	AR2sDSCv_UldConfirmBasketInfo[1,3].bAvailibility				:BOOL;

	(*Output Basket Counter*)*)
	(*diTotalBasketQty_Customer								:INT;*)


	bBasketQuality: BOOL;		(*Basket Quality identification- Good= True; Bad= False*)
(*Alarm*)
(*---------------------------------------------------------------------------------------------------------------------------------------------------------------------------------------------------------------------------------------------------------------------*)

(*ARbAlarmOutput-using global alarm*)

(*Recipe*)
(*----------------------------------------------------------------------------------------------------------------------------------------------------------------------------------------------------------------------------------------------------------------------------*)

	(*PPChangeStatus*)
	iSecsGemPPchange 		:INT;		(*Update Secs/Gem that PLC already create/Edit/Delete the recipe
											PPChangeStatus - Action done by PLC (0-Idle, 1-Created, 2-Edited, 3-Deleted)*)
	iSecsGemPPchangeName	:INT;			(*PPChangeName - Selected recipe*)

	(*PPExecName*)
	(*AR2sDSCv_LdConfirmBasketInfo[1,1].iProductRecipeNo*)         (*Update Secs/Gem the selected recipe to run the current basket*)

	(*PP-SelectName-server send Product No if the Remote Host is Enable/ON*)
	iServerSecsGemProgNo		:INT;


	(*HMI_Function.iRecipeNoFeed	-(Server Monitor), iServerSecsGemProgNo-(From server)  :INT;	(*During Online Remote Mode (PP-SELECT), Secs/Gem order machine to run this recipe*)*)

	(*PPDirectory*)
	sRecipeFileDirectory			:STRING(200);	(*Share folder for PLC to output all recipes. Collect the persistent data and configuration file from the Boot folder ?C:\TwinCAT\Boot*)

	(*PPUpdateStatus*)
	iSecsGemPPupdate		:INT;		(*Secs/Gem to inform PLC that specific recipe is already downloaded
										PPUpdateStatus - (0-Idle, 1-Created, 2-Edited, 3-Deleted)-once the file overwite is complete, SecsGem will write '2' to the Address. Use the same address (iSecsGemWriteCompleted)*)
	iSecsGemPPupdateName	:INT;		(*PPUpdateName - Selected recipe*)

	(*PPLog*)
	sSecsGemRecipeWriteLog		:ARRAY [0..4] OF STRING(200);	(*LabView will log 5 udated recipe event for PLC (to display at PLC)*)







END_VAR

// ---- GVLs/Secs_Gem/Global_Variables_Secs_Gem_Persistent.TcGVL
{attribute 'Tc2GvlVarNames'}
VAR_GLOBAL PERSISTENT


	iSecs_Control_State :INT;	(* Determine in Gem Console. Machine react base on this setting
							3 - Offline (Secs/GEM Offline - Remote Command disable)
							4 - Online Local (Secs/GEM Online - Local Control - Remote Command disable)
							5 - Online Remote (Secs/Gem Online - Host Control - Remote Command enable)*)

END_VAR

// ---- GVLs/SevenDay_Ctrl/Global_Variables_Process_Door.TcGVL
{attribute 'Tc2GvlVarNames'}
VAR_GLOBAL

(* xxxxxxxxxxxxxxxxxxxxxxxxxxxxxxxx Ld Door Variable xxxxxxxxxxxxxxxxxxxxxxxxxxxxxxxx*)
(*========================================================================*)

	wLdDoorOpen									: WORD;
	bLdDoorOpen_00									: BOOL;
	bLdDoorOpen_01									: BOOL;
	bLdDoorOpen_02									: BOOL;
	bLdDoorOpen_03									: BOOL;
	bLdDoorOpen_04									: BOOL;
	bLdDoorOpen_05									: BOOL;
	bLdDoorOpen_06									: BOOL;
	bLdDoorOpen_07									: BOOL;
	bLdDoorOpen_08									: BOOL;
	bLdDoorOpen_09									: BOOL;
	bLdDoorOpen_10									: BOOL;
	bLdDoorOpen_11									: BOOL;
	bLdDoorOpen_12									: BOOL;
	bLdDoorOpen_13									: BOOL;
	bLdDoorOpen_14									: BOOL;
	bLdDoorOpen_15									: BOOL;

	wLdDoorClose									: WORD;
	bLdDoorClose_00									: BOOL;
	bLdDoorClose_01									: BOOL;
	bLdDoorClose_02									: BOOL;
	bLdDoorClose_03									: BOOL;
	bLdDoorClose_04									: BOOL;
	bLdDoorClose_05									: BOOL;
	bLdDoorClose_06									: BOOL;
	bLdDoorClose_07									: BOOL;
	bLdDoorClose_08									: BOOL;
	bLdDoorClose_09									: BOOL;
	bLdDoorClose_10									: BOOL;
	bLdDoorClose_11									: BOOL;
	bLdDoorClose_12									: BOOL;
	bLdDoorClose_13									: BOOL;
	bLdDoorClose_14									: BOOL;
	bLdDoorClose_15									: BOOL;

	bLdDoorOpenCompleted							: BOOL;
	bLdDoorCloseCompleted							: BOOL;

	bLdDoorOpenAct									: BOOL;
	bLdDoorCloseAct									: BOOL;

(*HoldingBitSV*)

	bLdDoorOpenHolding								: BOOL;
	bLdDoorCloseHolding								: BOOL;
	bLdDoorClampHolding								: BOOL;
	bLdDoorUnClampHolding							: BOOL;

(* xxxxxxxxxxxxxxxxxxxxxxxxxxxxxxxx Stn1 Door Variable xxxxxxxxxxxxxxxxxxxxxxxxxxxxxxxx*)
(*========================================================================*)

	wStn1DoorOpen										: WORD;
	bStn1DoorOpen_00									: BOOL;
	bStn1DoorOpen_01									: BOOL;
	bStn1DoorOpen_02									: BOOL;
	bStn1DoorOpen_03									: BOOL;
	bStn1DoorOpen_04									: BOOL;
	bStn1DoorOpen_05									: BOOL;
	bStn1DoorOpen_06									: BOOL;
	bStn1DoorOpen_07									: BOOL;
	bStn1DoorOpen_08									: BOOL;
	bStn1DoorOpen_09									: BOOL;
	bStn1DoorOpen_10									: BOOL;
	bStn1DoorOpen_11									: BOOL;
	bStn1DoorOpen_12									: BOOL;
	bStn1DoorOpen_13									: BOOL;
	bStn1DoorOpen_14									: BOOL;
	bStn1DoorOpen_15									: BOOL;

	wStn1DoorClose										: WORD;
	bStn1DoorClose_00									: BOOL;
	bStn1DoorClose_01									: BOOL;
	bStn1DoorClose_02									: BOOL;
	bStn1DoorClose_03									: BOOL;
	bStn1DoorClose_04									: BOOL;
	bStn1DoorClose_05									: BOOL;
	bStn1DoorClose_06									: BOOL;
	bStn1DoorClose_07									: BOOL;
	bStn1DoorClose_08									: BOOL;
	bStn1DoorClose_09									: BOOL;
	bStn1DoorClose_10									: BOOL;
	bStn1DoorClose_11									: BOOL;
	bStn1DoorClose_12									: BOOL;
	bStn1DoorClose_13									: BOOL;
	bStn1DoorClose_14									: BOOL;
	bStn1DoorClose_15									: BOOL;

	bStn1DoorOpenCompleted								: BOOL;
	bStn1DoorCloseCompleted								: BOOL;

	bStn1DoorOpenAct									: BOOL;
	bStn1DoorCloseAct									: BOOL;

(*HoldingBitSV*)

	bStn1DoorOpenHolding								: BOOL;
	bStn1DoorCloseHolding								: BOOL;
	bStn1DoorClampHolding								: BOOL;
	bStn1DoorUnClampHolding								: BOOL;

(* xxxxxxxxxxxxxxxxxxxxxxxxxxxxxxxx Stn2 Door Variable xxxxxxxxxxxxxxxxxxxxxxxxxxxxxxxx*)
(*========================================================================*)

	wStn2DoorOpen										: WORD;
	bStn2DoorOpen_00									: BOOL;
	bStn2DoorOpen_01									: BOOL;
	bStn2DoorOpen_02									: BOOL;
	bStn2DoorOpen_03									: BOOL;
	bStn2DoorOpen_04									: BOOL;
	bStn2DoorOpen_05									: BOOL;
	bStn2DoorOpen_06									: BOOL;
	bStn2DoorOpen_07									: BOOL;
	bStn2DoorOpen_08									: BOOL;
	bStn2DoorOpen_09									: BOOL;
	bStn2DoorOpen_10									: BOOL;
	bStn2DoorOpen_11									: BOOL;
	bStn2DoorOpen_12									: BOOL;
	bStn2DoorOpen_13									: BOOL;
	bStn2DoorOpen_14									: BOOL;
	bStn2DoorOpen_15									: BOOL;

	wStn2DoorClose										: WORD;
	bStn2DoorClose_00									: BOOL;
	bStn2DoorClose_01									: BOOL;
	bStn2DoorClose_02									: BOOL;
	bStn2DoorClose_03									: BOOL;
	bStn2DoorClose_04									: BOOL;
	bStn2DoorClose_05									: BOOL;
	bStn2DoorClose_06									: BOOL;
	bStn2DoorClose_07									: BOOL;
	bStn2DoorClose_08									: BOOL;
	bStn2DoorClose_09									: BOOL;
	bStn2DoorClose_10									: BOOL;
	bStn2DoorClose_11									: BOOL;
	bStn2DoorClose_12									: BOOL;
	bStn2DoorClose_13									: BOOL;
	bStn2DoorClose_14									: BOOL;
	bStn2DoorClose_15									: BOOL;

	bStn2DoorOpenCompleted								: BOOL;
	bStn2DoorCloseCompleted								: BOOL;

	bStn2DoorOpenAct									: BOOL;
	bStn2DoorCloseAct									: BOOL;

(*HoldingBitSV*)

	bStn2DoorOpenHolding								: BOOL;
	bStn2DoorCloseHolding								: BOOL;
	bStn2DoorClampHolding								: BOOL;
	bStn2DoorUnClampHolding								: BOOL;

(* xxxxxxxxxxxxxxxxxxxxxxxxxxxxxxxx Stn3 Door Variable xxxxxxxxxxxxxxxxxxxxxxxxxxxxxxxx*)
(*========================================================================*)

	wStn3DoorOpen										: WORD;
	bStn3DoorOpen_00									: BOOL;
	bStn3DoorOpen_01									: BOOL;
	bStn3DoorOpen_02									: BOOL;
	bStn3DoorOpen_03									: BOOL;
	bStn3DoorOpen_04									: BOOL;
	bStn3DoorOpen_05									: BOOL;
	bStn3DoorOpen_06									: BOOL;
	bStn3DoorOpen_07									: BOOL;
	bStn3DoorOpen_08									: BOOL;
	bStn3DoorOpen_09									: BOOL;
	bStn3DoorOpen_10									: BOOL;
	bStn3DoorOpen_11									: BOOL;
	bStn3DoorOpen_12									: BOOL;
	bStn3DoorOpen_13									: BOOL;
	bStn3DoorOpen_14									: BOOL;
	bStn3DoorOpen_15									: BOOL;

	wStn3DoorClose										: WORD;
	bStn3DoorClose_00									: BOOL;
	bStn3DoorClose_01									: BOOL;
	bStn3DoorClose_02									: BOOL;
	bStn3DoorClose_03									: BOOL;
	bStn3DoorClose_04									: BOOL;
	bStn3DoorClose_05									: BOOL;
	bStn3DoorClose_06									: BOOL;
	bStn3DoorClose_07									: BOOL;
	bStn3DoorClose_08									: BOOL;
	bStn3DoorClose_09									: BOOL;
	bStn3DoorClose_10									: BOOL;
	bStn3DoorClose_11									: BOOL;
	bStn3DoorClose_12									: BOOL;
	bStn3DoorClose_13									: BOOL;
	bStn3DoorClose_14									: BOOL;
	bStn3DoorClose_15									: BOOL;

	bStn3DoorOpenCompleted								: BOOL;
	bStn3DoorCloseCompleted								: BOOL;

	bStn3DoorOpenAct									: BOOL;
	bStn3DoorCloseAct									: BOOL;

(*HoldingBitSV*)

	bStn3DoorOpenHolding								: BOOL;
	bStn3DoorCloseHolding								: BOOL;
	bStn3DoorClampHolding								: BOOL;
	bStn3DoorUnClampHolding								: BOOL;

(* xxxxxxxxxxxxxxxxxxxxxxxxxxxxxxxx Stn4 Door Variable xxxxxxxxxxxxxxxxxxxxxxxxxxxxxxxx*)
(*========================================================================*)

	wStn4DoorOpen										: WORD;
	bStn4DoorOpen_00									: BOOL;
	bStn4DoorOpen_01									: BOOL;
	bStn4DoorOpen_02									: BOOL;
	bStn4DoorOpen_03									: BOOL;
	bStn4DoorOpen_04									: BOOL;
	bStn4DoorOpen_05									: BOOL;
	bStn4DoorOpen_06									: BOOL;
	bStn4DoorOpen_07									: BOOL;
	bStn4DoorOpen_08									: BOOL;
	bStn4DoorOpen_09									: BOOL;
	bStn4DoorOpen_10									: BOOL;
	bStn4DoorOpen_11									: BOOL;
	bStn4DoorOpen_12									: BOOL;
	bStn4DoorOpen_13									: BOOL;
	bStn4DoorOpen_14									: BOOL;
	bStn4DoorOpen_15									: BOOL;

	wStn4DoorClose										: WORD;
	bStn4DoorClose_00									: BOOL;
	bStn4DoorClose_01									: BOOL;
	bStn4DoorClose_02									: BOOL;
	bStn4DoorClose_03									: BOOL;
	bStn4DoorClose_04									: BOOL;
	bStn4DoorClose_05									: BOOL;
	bStn4DoorClose_06									: BOOL;
	bStn4DoorClose_07									: BOOL;
	bStn4DoorClose_08									: BOOL;
	bStn4DoorClose_09									: BOOL;
	bStn4DoorClose_10									: BOOL;
	bStn4DoorClose_11									: BOOL;
	bStn4DoorClose_12									: BOOL;
	bStn4DoorClose_13									: BOOL;
	bStn4DoorClose_14									: BOOL;
	bStn4DoorClose_15									: BOOL;

	bStn4DoorOpenCompleted								: BOOL;
	bStn4DoorCloseCompleted								: BOOL;

	bStn4DoorOpenAct									: BOOL;
	bStn4DoorCloseAct									: BOOL;

(*HoldingBitSV*)

	bStn4DoorOpenHolding								: BOOL;
	bStn4DoorCloseHolding								: BOOL;
	bStn4DoorClampHolding								: BOOL;
	bStn4DoorUnClampHolding								: BOOL;

(* xxxxxxxxxxxxxxxxxxxxxxxxxxxxxxxx Stn5 Door Variable xxxxxxxxxxxxxxxxxxxxxxxxxxxxxxxx*)
(*========================================================================*)

	wStn5DoorOpen										: WORD;
	bStn5DoorOpen_00									: BOOL;
	bStn5DoorOpen_01									: BOOL;
	bStn5DoorOpen_02									: BOOL;
	bStn5DoorOpen_03									: BOOL;
	bStn5DoorOpen_04									: BOOL;
	bStn5DoorOpen_05									: BOOL;
	bStn5DoorOpen_06									: BOOL;
	bStn5DoorOpen_07									: BOOL;
	bStn5DoorOpen_08									: BOOL;
	bStn5DoorOpen_09									: BOOL;
	bStn5DoorOpen_10									: BOOL;
	bStn5DoorOpen_11									: BOOL;
	bStn5DoorOpen_12									: BOOL;
	bStn5DoorOpen_13									: BOOL;
	bStn5DoorOpen_14									: BOOL;
	bStn5DoorOpen_15									: BOOL;

	wStn5DoorClose										: WORD;
	bStn5DoorClose_00									: BOOL;
	bStn5DoorClose_01									: BOOL;
	bStn5DoorClose_02									: BOOL;
	bStn5DoorClose_03									: BOOL;
	bStn5DoorClose_04									: BOOL;
	bStn5DoorClose_05									: BOOL;
	bStn5DoorClose_06									: BOOL;
	bStn5DoorClose_07									: BOOL;
	bStn5DoorClose_08									: BOOL;
	bStn5DoorClose_09									: BOOL;
	bStn5DoorClose_10									: BOOL;
	bStn5DoorClose_11									: BOOL;
	bStn5DoorClose_12									: BOOL;
	bStn5DoorClose_13									: BOOL;
	bStn5DoorClose_14									: BOOL;
	bStn5DoorClose_15									: BOOL;

	bStn5DoorOpenCompleted								: BOOL;
	bStn5DoorCloseCompleted								: BOOL;

	bStn5DoorOpenAct									: BOOL;
	bStn5DoorCloseAct									: BOOL;

(*HoldingBitSV*)

	bStn5DoorOpenHolding								: BOOL;
	bStn5DoorCloseHolding								: BOOL;
	bStn5DoorClampHolding								: BOOL;
	bStn5DoorUnClampHolding								: BOOL;

(* xxxxxxxxxxxxxxxxxxxxxxxxxxxxxxxx Stn6 Door Variable xxxxxxxxxxxxxxxxxxxxxxxxxxxxxxxx*)
(*========================================================================*)

	wStn6DoorOpen										: WORD;
	bStn6DoorOpen_00									: BOOL;
	bStn6DoorOpen_01									: BOOL;
	bStn6DoorOpen_02									: BOOL;
	bStn6DoorOpen_03									: BOOL;
	bStn6DoorOpen_04									: BOOL;
	bStn6DoorOpen_05									: BOOL;
	bStn6DoorOpen_06									: BOOL;
	bStn6DoorOpen_07									: BOOL;
	bStn6DoorOpen_08									: BOOL;
	bStn6DoorOpen_09									: BOOL;
	bStn6DoorOpen_10									: BOOL;
	bStn6DoorOpen_11									: BOOL;
	bStn6DoorOpen_12									: BOOL;
	bStn6DoorOpen_13									: BOOL;
	bStn6DoorOpen_14									: BOOL;
	bStn6DoorOpen_15									: BOOL;

	wStn6DoorClose										: WORD;
	bStn6DoorClose_00									: BOOL;
	bStn6DoorClose_01									: BOOL;
	bStn6DoorClose_02									: BOOL;
	bStn6DoorClose_03									: BOOL;
	bStn6DoorClose_04									: BOOL;
	bStn6DoorClose_05									: BOOL;
	bStn6DoorClose_06									: BOOL;
	bStn6DoorClose_07									: BOOL;
	bStn6DoorClose_08									: BOOL;
	bStn6DoorClose_09									: BOOL;
	bStn6DoorClose_10									: BOOL;
	bStn6DoorClose_11									: BOOL;
	bStn6DoorClose_12									: BOOL;
	bStn6DoorClose_13									: BOOL;
	bStn6DoorClose_14									: BOOL;
	bStn6DoorClose_15									: BOOL;

	bStn6DoorOpenCompleted								: BOOL;
	bStn6DoorCloseCompleted								: BOOL;

	bStn6DoorOpenAct									: BOOL;
	bStn6DoorCloseAct									: BOOL;

(*HoldingBitSV*)

	bStn6DoorOpenHolding								: BOOL;
	bStn6DoorCloseHolding								: BOOL;
	bStn6DoorClampHolding								: BOOL;
	bStn6DoorUnClampHolding								: BOOL;

(* xxxxxxxxxxxxxxxxxxxxxxxxxxxxxxxx Stn7 Door Variable xxxxxxxxxxxxxxxxxxxxxxxxxxxxxxxx*)
(*========================================================================*)

	wStn7DoorOpen										: WORD;
	bStn7DoorOpen_00									: BOOL;
	bStn7DoorOpen_01									: BOOL;
	bStn7DoorOpen_02									: BOOL;
	bStn7DoorOpen_03									: BOOL;
	bStn7DoorOpen_04									: BOOL;
	bStn7DoorOpen_05									: BOOL;
	bStn7DoorOpen_06									: BOOL;
	bStn7DoorOpen_07									: BOOL;
	bStn7DoorOpen_08									: BOOL;
	bStn7DoorOpen_09									: BOOL;
	bStn7DoorOpen_10									: BOOL;
	bStn7DoorOpen_11									: BOOL;
	bStn7DoorOpen_12									: BOOL;
	bStn7DoorOpen_13									: BOOL;
	bStn7DoorOpen_14									: BOOL;
	bStn7DoorOpen_15									: BOOL;

	wStn7DoorClose										: WORD;
	bStn7DoorClose_00									: BOOL;
	bStn7DoorClose_01									: BOOL;
	bStn7DoorClose_02									: BOOL;
	bStn7DoorClose_03									: BOOL;
	bStn7DoorClose_04									: BOOL;
	bStn7DoorClose_05									: BOOL;
	bStn7DoorClose_06									: BOOL;
	bStn7DoorClose_07									: BOOL;
	bStn7DoorClose_08									: BOOL;
	bStn7DoorClose_09									: BOOL;
	bStn7DoorClose_10									: BOOL;
	bStn7DoorClose_11									: BOOL;
	bStn7DoorClose_12									: BOOL;
	bStn7DoorClose_13									: BOOL;
	bStn7DoorClose_14									: BOOL;
	bStn7DoorClose_15									: BOOL;

	bStn7DoorOpenCompleted								: BOOL;
	bStn7DoorCloseCompleted								: BOOL;

	bStn7DoorOpenAct									: BOOL;
	bStn7DoorCloseAct									: BOOL;

(*HoldingitSV*)

	bStn7DoorOpenHolding								: BOOL;
	bStn7DoorCloseHolding								: BOOL;
	bStn7DoorClampHolding								: BOOL;
	bStn7DoorUnClampHolding								: BOOL;

(* xxxxxxxxxxxxxxxxxxxxxxxxxxxxxxxx Stn8 Door Variable xxxxxxxxxxxxxxxxxxxxxxxxxxxxxxxx*)
(*========================================================================*)

	wStn8DoorOpen										: WORD;
	bStn8DoorOpen_00									: BOOL;
	bStn8DoorOpen_01									: BOOL;
	bStn8DoorOpen_02									: BOOL;
	bStn8DoorOpen_03									: BOOL;
	bStn8DoorOpen_04									: BOOL;
	bStn8DoorOpen_05									: BOOL;
	bStn8DoorOpen_06									: BOOL;
	bStn8DoorOpen_07									: BOOL;
	bStn8DoorOpen_08									: BOOL;
	bStn8DoorOpen_09									: BOOL;
	bStn8DoorOpen_10									: BOOL;
	bStn8DoorOpen_11									: BOOL;
	bStn8DoorOpen_12									: BOOL;
	bStn8DoorOpen_13									: BOOL;
	bStn8DoorOpen_14									: BOOL;
	bStn8DoorOpen_15									: BOOL;

	wStn8DoorClose										: WORD;
	bStn8DoorClose_00									: BOOL;
	bStn8DoorClose_01									: BOOL;
	bStn8DoorClose_02									: BOOL;
	bStn8DoorClose_03									: BOOL;
	bStn8DoorClose_04									: BOOL;
	bStn8DoorClose_05									: BOOL;
	bStn8DoorClose_06									: BOOL;
	bStn8DoorClose_07									: BOOL;
	bStn8DoorClose_08									: BOOL;
	bStn8DoorClose_09									: BOOL;
	bStn8DoorClose_10									: BOOL;
	bStn8DoorClose_11									: BOOL;
	bStn8DoorClose_12									: BOOL;
	bStn8DoorClose_13									: BOOL;
	bStn8DoorClose_14									: BOOL;
	bStn8DoorClose_15									: BOOL;

	bStn8DoorOpenCompleted								: BOOL;
	bStn8DoorCloseCompleted								: BOOL;

	bStn8DoorOpenAct									: BOOL;
	bStn8DoorCloseAct									: BOOL;

(*HoldingBitSV*)

	bStn8DoorOpenHolding								: BOOL;
	bStn8DoorCloseHolding								: BOOL;
	bStn8DoorClampHolding								: BOOL;
	bStn8DoorUnClampHolding								: BOOL;

(* xxxxxxxxxxxxxxxxxxxxxxxxxxxxxxxx Stn9 Door Variable xxxxxxxxxxxxxxxxxxxxxxxxxxxxxxxx*)
(*========================================================================*)

	wStn9DoorOpen										: WORD;
	bStn9DoorOpen_00									: BOOL;
	bStn9DoorOpen_01									: BOOL;
	bStn9DoorOpen_02									: BOOL;
	bStn9DoorOpen_03									: BOOL;
	bStn9DoorOpen_04									: BOOL;
	bStn9DoorOpen_05									: BOOL;
	bStn9DoorOpen_06									: BOOL;
	bStn9DoorOpen_07									: BOOL;
	bStn9DoorOpen_08									: BOOL;
	bStn9DoorOpen_09									: BOOL;
	bStn9DoorOpen_10									: BOOL;
	bStn9DoorOpen_11									: BOOL;
	bStn9DoorOpen_12									: BOOL;
	bStn9DoorOpen_13									: BOOL;
	bStn9DoorOpen_14									: BOOL;
	bStn9DoorOpen_15									: BOOL;

	wStn9DoorClose										: WORD;
	bStn9DoorClose_00									: BOOL;
	bStn9DoorClose_01									: BOOL;
	bStn9DoorClose_02									: BOOL;
	bStn9DoorClose_03									: BOOL;
	bStn9DoorClose_04									: BOOL;
	bStn9DoorClose_05									: BOOL;
	bStn9DoorClose_06									: BOOL;
	bStn9DoorClose_07									: BOOL;
	bStn9DoorClose_08									: BOOL;
	bStn9DoorClose_09									: BOOL;
	bStn9DoorClose_10									: BOOL;
	bStn9DoorClose_11									: BOOL;
	bStn9DoorClose_12									: BOOL;
	bStn9DoorClose_13									: BOOL;
	bStn9DoorClose_14									: BOOL;
	bStn9DoorClose_15									: BOOL;

	bStn9DoorOpenCompleted								: BOOL;
	bStn9DoorCloseCompleted								: BOOL;

	bStn9DoorOpenAct									: BOOL;
	bStn9DoorCloseAct									: BOOL;

(*HoldingBitSV*)

	bStn9DoorOpenHolding								: BOOL;
	bStn9DoorCloseHolding								: BOOL;
	bStn9DoorClampHolding								: BOOL;
	bStn9DoorUnClampHolding								: BOOL;

(* xxxxxxxxxxxxxxxxxxxxxxxxxxxxxxxx Stn10 Door Variable xxxxxxxxxxxxxxxxxxxxxxxxxxxxxxxx*)
(*========================================================================*)

	wStn10DoorOpen										: WORD;
	bStn10DoorOpen_00									: BOOL;
	bStn10DoorOpen_01									: BOOL;
	bStn10DoorOpen_02									: BOOL;
	bStn10DoorOpen_03									: BOOL;
	bStn10DoorOpen_04									: BOOL;
	bStn10DoorOpen_05									: BOOL;
	bStn10DoorOpen_06									: BOOL;
	bStn10DoorOpen_07									: BOOL;
	bStn10DoorOpen_08									: BOOL;
	bStn10DoorOpen_09									: BOOL;
	bStn10DoorOpen_10									: BOOL;
	bStn10DoorOpen_11									: BOOL;
	bStn10DoorOpen_12									: BOOL;
	bStn10DoorOpen_13									: BOOL;
	bStn10DoorOpen_14									: BOOL;
	bStn10DoorOpen_15									: BOOL;

	wStn10DoorClose										: WORD;
	bStn10DoorClose_00									: BOOL;
	bStn10DoorClose_01									: BOOL;
	bStn10DoorClose_02									: BOOL;
	bStn10DoorClose_03									: BOOL;
	bStn10DoorClose_04									: BOOL;
	bStn10DoorClose_05									: BOOL;
	bStn10DoorClose_06									: BOOL;
	bStn10DoorClose_07									: BOOL;
	bStn10DoorClose_08									: BOOL;
	bStn10DoorClose_09									: BOOL;
	bStn10DoorClose_10									: BOOL;
	bStn10DoorClose_11									: BOOL;
	bStn10DoorClose_12									: BOOL;
	bStn10DoorClose_13									: BOOL;
	bStn10DoorClose_14									: BOOL;
	bStn10DoorClose_15									: BOOL;

	bStn10DoorOpenCompleted							: BOOL;
	bStn10DoorCloseCompleted							: BOOL;

	bStn10DoorOpenAct									: BOOL;
	bStn10DoorCloseAct									: BOOL;

(*HoldingBitSV*)

	bStn10DoorOpenHolding								: BOOL;
	bStn10DoorCloseHolding								: BOOL;
	bStn10DoorClampHolding								: BOOL;
	bStn10DoorUnClampHolding							: BOOL;

(* xxxxxxxxxxxxxxxxxxxxxxxxxxxxxxxx Stn11 Door Variable xxxxxxxxxxxxxxxxxxxxxxxxxxxxxxxx*)
(*========================================================================*)

	wStn11DoorOpen										: WORD;
	bStn11DoorOpen_00									: BOOL;
	bStn11DoorOpen_01									: BOOL;
	bStn11DoorOpen_02									: BOOL;
	bStn11DoorOpen_03									: BOOL;
	bStn11DoorOpen_04									: BOOL;
	bStn11DoorOpen_05									: BOOL;
	bStn11DoorOpen_06									: BOOL;
	bStn11DoorOpen_07									: BOOL;
	bStn11DoorOpen_08									: BOOL;
	bStn11DoorOpen_09									: BOOL;
	bStn11DoorOpen_10									: BOOL;
	bStn11DoorOpen_11									: BOOL;
	bStn11DoorOpen_12									: BOOL;
	bStn11DoorOpen_13									: BOOL;
	bStn11DoorOpen_14									: BOOL;
	bStn11DoorOpen_15									: BOOL;

	wStn11DoorClose										: WORD;
	bStn11DoorClose_00									: BOOL;
	bStn11DoorClose_01									: BOOL;
	bStn11DoorClose_02									: BOOL;
	bStn11DoorClose_03									: BOOL;
	bStn11DoorClose_04									: BOOL;
	bStn11DoorClose_05									: BOOL;
	bStn11DoorClose_06									: BOOL;
	bStn11DoorClose_07									: BOOL;
	bStn11DoorClose_08									: BOOL;
	bStn11DoorClose_09									: BOOL;
	bStn11DoorClose_10									: BOOL;
	bStn11DoorClose_11									: BOOL;
	bStn11DoorClose_12									: BOOL;
	bStn11DoorClose_13									: BOOL;
	bStn11DoorClose_14									: BOOL;
	bStn11DoorClose_15									: BOOL;

	bStn11DoorOpenCompleted							: BOOL;
	bStn11DoorCloseCompleted							: BOOL;

	bStn11DoorOpenAct									: BOOL;
	bStn11DoorCloseAct									: BOOL;

(*HoldingBitSV*)

	bStn11DoorOpenHolding								: BOOL;
	bStn11DoorCloseHolding								: BOOL;
	bStn11DoorClampHolding								: BOOL;
	bStn11DoorUnClampHolding							: BOOL;

(* xxxxxxxxxxxxxxxxxxxxxxxxxxxxxxxx Stn12 Door Variable xxxxxxxxxxxxxxxxxxxxxxxxxxxxxxxx*)
(*========================================================================*)

	wStn12DoorOpen										: WORD;
	bStn12DoorOpen_00									: BOOL;
	bStn12DoorOpen_01									: BOOL;
	bStn12DoorOpen_02									: BOOL;
	bStn12DoorOpen_03									: BOOL;
	bStn12DoorOpen_04									: BOOL;
	bStn12DoorOpen_05									: BOOL;
	bStn12DoorOpen_06									: BOOL;
	bStn12DoorOpen_07									: BOOL;
	bStn12DoorOpen_08									: BOOL;
	bStn12DoorOpen_09									: BOOL;
	bStn12DoorOpen_10									: BOOL;
	bStn12DoorOpen_11									: BOOL;
	bStn12DoorOpen_12									: BOOL;
	bStn12DoorOpen_13									: BOOL;
	bStn12DoorOpen_14									: BOOL;
	bStn12DoorOpen_15									: BOOL;

	wStn12DoorClose										: WORD;
	bStn12DoorClose_00									: BOOL;
	bStn12DoorClose_01									: BOOL;
	bStn12DoorClose_02									: BOOL;
	bStn12DoorClose_03									: BOOL;
	bStn12DoorClose_04									: BOOL;
	bStn12DoorClose_05									: BOOL;
	bStn12DoorClose_06									: BOOL;
	bStn12DoorClose_07									: BOOL;
	bStn12DoorClose_08									: BOOL;
	bStn12DoorClose_09									: BOOL;
	bStn12DoorClose_10									: BOOL;
	bStn12DoorClose_11									: BOOL;
	bStn12DoorClose_12									: BOOL;
	bStn12DoorClose_13									: BOOL;
	bStn12DoorClose_14									: BOOL;
	bStn12DoorClose_15									: BOOL;

	bStn12DoorOpenCompleted							: BOOL;
	bStn12DoorCloseCompleted							: BOOL;

	bStn12DoorOpenAct									: BOOL;
	bStn12DoorCloseAct									: BOOL;

(*HoldingBitSV*)

	bStn12DoorOpenHolding								: BOOL;
	bStn12DoorCloseHolding								: BOOL;
	bStn12DoorClampHolding								: BOOL;
	bStn12DoorUnClampHolding							: BOOL;

(* xxxxxxxxxxxxxxxxxxxxxxxxxxxxxxxx Uld Door Variable xxxxxxxxxxxxxxxxxxxxxxxxxxxxxxxx*)
(*========================================================================*)

	wUldDoorOpen										: WORD;
	bUldDoorOpen_00										: BOOL;
	bUldDoorOpen_01										: BOOL;
	bUldDoorOpen_02										: BOOL;
	bUldDoorOpen_03										: BOOL;
	bUldDoorOpen_04										: BOOL;
	bUldDoorOpen_05										: BOOL;
	bUldDoorOpen_06										: BOOL;
	bUldDoorOpen_07										: BOOL;
	bUldDoorOpen_08										: BOOL;
	bUldDoorOpen_09										: BOOL;
	bUldDoorOpen_10										: BOOL;
	bUldDoorOpen_11										: BOOL;
	bUldDoorOpen_12										: BOOL;
	bUldDoorOpen_13										: BOOL;
	bUldDoorOpen_14										: BOOL;
	bUldDoorOpen_15										: BOOL;

	wUldDoorClose										: WORD;
	bUldDoorClose_00									: BOOL;
	bUldDoorClose_01									: BOOL;
	bUldDoorClose_02									: BOOL;
	bUldDoorClose_03									: BOOL;
	bUldDoorClose_04									: BOOL;
	bUldDoorClose_05									: BOOL;
	bUldDoorClose_06									: BOOL;
	bUldDoorClose_07									: BOOL;
	bUldDoorClose_08									: BOOL;
	bUldDoorClose_09									: BOOL;
	bUldDoorClose_10									: BOOL;
	bUldDoorClose_11									: BOOL;
	bUldDoorClose_12									: BOOL;
	bUldDoorClose_13									: BOOL;
	bUldDoorClose_14									: BOOL;
	bUldDoorClose_15									: BOOL;

	bUldDoorOpenCompleted								: BOOL;
	bUldDoorCloseCompleted								: BOOL;

	bUldDoorOpenAct										: BOOL;
	bUldDoorCloseAct									: BOOL;

(*HoldingBitSV*)

	bUldDoorOpenHolding									: BOOL;
	bUldDoorCloseHolding								: BOOL;
	bUldDoorClampHolding								: BOOL;
	bUldDoorUnClampHolding								: BOOL;

	bUldTransferInHolding									: BOOL;
	bUldTransferOutHolding								: BOOL;


(*Conveyor holding*)


	bLdConveyorPopupInHolding							: BOOL;
	bLdConveyorPopupOutHolding							: BOOL;
	bUldConveyorPopupInHolding							: BOOL;
	bUldConveyorPopupOutHolding							: BOOL;

	bLdConveyorUpHolding								: BOOL;
	bLdConveyorDownHolding								: BOOL;
	bUldConveyorUpHolding								: BOOL;
	bUldConveyorDownHolding								: BOOL;

	bLdConveyorPusherInHolding							: BOOL;
	bLdConveyorPusherOutHolding							: BOOL;
	bUldConveyorPusherInHolding							: BOOL;
	bUldConveyorPusherOutHolding						: BOOL;
	
	bUldConveyorOpenHolding								: BOOL;
	bUldConveyorCloseHolding							: BOOL;
	
	wUldConveyorOpen									: WORD;	
	bUldConveyorOpen_00									: BOOL;
	bUldConveyorOpen_01									: BOOL;
	bUldConveyorOpen_02									: BOOL;
	bUldConveyorOpen_03									: BOOL;
	bUldConveyorOpen_04									: BOOL;
	bUldConveyorOpen_05									: BOOL;
	bUldConveyorOpen_06									: BOOL;
	bUldConveyorOpen_07									: BOOL;
	bUldConveyorOpen_08									: BOOL;
	bUldConveyorOpen_09									: BOOL;
	bUldConveyorOpen_10									: BOOL;
	bUldConveyorOpen_11									: BOOL;
	bUldConveyorOpen_12									: BOOL;
	bUldConveyorOpen_13									: BOOL;
	bUldConveyorOpen_14									: BOOL;
	bUldConveyorOpen_15									: BOOL;

	wUldConveyorClose									: WORD;
	bUldConveyorClose_00								: BOOL;
	bUldConveyorClose_01								: BOOL;
	bUldConveyorClose_02								: BOOL;
	bUldConveyorClose_03								: BOOL;
	bUldConveyorClose_04								: BOOL;
	bUldConveyorClose_05								: BOOL;
	bUldConveyorClose_06								: BOOL;
	bUldConveyorClose_07								: BOOL;
	bUldConveyorClose_08								: BOOL;
	bUldConveyorClose_09								: BOOL;
	bUldConveyorClose_10								: BOOL;
	bUldConveyorClose_11								: BOOL;
	bUldConveyorClose_12								: BOOL;
	bUldConveyorClose_13								: BOOL;
	bUldConveyorClose_14								: BOOL;
	bUldConveyorClose_15								: BOOL;

	
	bUldConveyorOpenCompleted							: BOOL;
	bUldConveyorCloseCompleted							: BOOL;
	
	

(*StnCylinderReciprocating*)

	bStnCylinderReciprocating								: BOOL;

END_VAR

// ---- GVLs/SevenDay_Ctrl/Global_Variables_SevenDay_NoPersistent.TcGVL
{attribute 'Tc2GvlVarNames'}
VAR_GLOBAL

	bAutoSysOn			: BOOL;
	bSevenDaySysOn 	: BOOL;
	bSevenDaySysOff 	: BOOL;

END_VAR

// ---- GVLs/SevenDay_Ctrl/Global_Variables_SevenDay_Persistent.TcGVL
{attribute 'Tc2GvlVarNames'}
VAR_GLOBAL PERSISTENT

	TodayDay 				: STRING;

	ArbDayOnEn_IN			: ARRAY [1..7] OF BOOL;
	ArbDayOffEn_IN			: ARRAY [1..7] OF BOOL;

	ArwDayOnHour_IN		: ARRAY [1..7] OF WORD;
	ArwDayOnMinute_IN		: ARRAY [1..7] OF WORD;

	ArwDayOffHour_IN		: ARRAY [1..7] OF WORD;
	ArwDayOffMinute_IN		: ARRAY [1..7] OF WORD;

	ArbDaySysOn_OUT		: ARRAY [1..7] OF BOOL;
	ArbDaySysOff_OUT		: ARRAY [1..7] OF BOOL;

END_VAR

// ---- GVLs/Special_Ctrl/Global_Variables_Special_NoPersistent.TcGVL
{attribute 'Tc2GvlVarNames'}
VAR_GLOBAL

(* xxxxxxxxxxxxxxxxxxxxxxxxxxxxxxxx Temperature Cltr xxxxxxxxxxxxxxxxxxxxxxxxxxxxxxxx*)
(*========================================================================*)

	ARrStnWaterJacketTempPV									: ARRAY [1..iStnQty] OF REAL;
	ARbStnWaterJacketTempOnOff									: ARRAY [1..iStnQty] OF BOOL;
	ARbStnWaterJacketTempRDY									: ARRAY [1..iStnQty] OF BOOL;
	ARbStnWaterJacketTempHAL									: ARRAY [1..iStnQty] OF BOOL;
	ARbStnWaterJacketTemp1stLimitAlarm							: ARRAY [1..iStnQty] OF BOOL;
	ARbStnWaterJacketTemp2ndLimitAlarm							: ARRAY [1..iStnQty] OF BOOL;
	ARbStnWaterJacketTempPreparationNoRdyAlarm					: ARRAY [1..iStnQty] OF BOOL;

	ARrStnSubTankTempPV											: ARRAY [1..iStnQty] OF REAL;
	ARbStnSubTankTempOnOff										: ARRAY [1..iStnQty] OF BOOL;
	ARbStnSubTankTempRDY										: ARRAY [1..iStnQty] OF BOOL;
	ARbStnSubTankTempHAL										: ARRAY [1..iStnQty] OF BOOL;
	ARbStnSubTankTemp1stLimitAlarm								: ARRAY [1..iStnQty] OF BOOL;
	ARbStnSubTankTemp2ndLimitAlarm								: ARRAY [1..iStnQty] OF BOOL;
	ARbStnSubTankTempPreparationNoRdyAlarm						: ARRAY [1..iStnQty] OF BOOL;

	rJRSInlineHeaterTempPV										: REAL;
	bJRSInlineHeaterTempOnOff									: BOOL;
	bJRSInlineHeaterTempRDY										: BOOL;
	bJRSInlineHeaterTempHAL										: BOOL;
	bJRSInlineHeaterTemp1stLimitAlarm							: BOOL;
	bJRSInlineHeaterTemp2ndLimitAlarm							: BOOL;
	bJRSInlineHeaterTempPreparationNoRdyAlarm					: BOOL;

	rIncTempPV													: REAL;
	bIncTempOnOff												: BOOL;
	bIncTempRDY													: BOOL;
	bIncTempHAL													: BOOL;
	bIncTemp1stLimitAlarm										: BOOL;
	bIncTemp2ndLimitAlarm										: BOOL;
	bIncTempPreparationNoRdyAlarm								: BOOL;

	rOilSeparatorTempPV											: REAL;
	bOilSeparatorTempOnOff										: BOOL;
	bOilSeparatorTempRDY										: BOOL;
	bOilSeparatorTempHAL										: BOOL;
	bOilSeparatorTemp1stLimitAlarm								: BOOL;
	bOilSeparatorTemp2ndLimitAlarm								: BOOL;
	bOilSeparatorTempPreparationNoRdyAlarm						: BOOL;
	
// 1= Left Top, 2 = Left Bottom, 3= Right Top, 4= Right bottom		
	ARrStnExternalTempPV										: ARRAY [1..4] OF  REAL;
	ARbStnExternalTempOnOff										: ARRAY [1..4] OF  BOOL;
	ARbStnExternalempRDY										: ARRAY [1..4] OF  BOOL;
	ARbStnExternalTempHAL										: ARRAY [1..4] OF  BOOL;
	ARbStnExternalTemp1stLimitAlarm								: ARRAY [1..4] OF  BOOL;
	ARbStnExternalTemp2ndLimitAlarm								: ARRAY [1..4] OF  BOOL;
	ARbStnExternalTempPreparationNoRdyAlarm						: ARRAY [1..4] OF  BOOL;

	ARrStnIncVaporPurgeTempPV									: ARRAY [1..iStnQty] OF REAL;
	
		rStnExternalTempMINsvHMIDisplay								: REAL;
	rStnExternalTempMAXsvHMIDisplay								: REAL;
	
	rStnExternalTempHALMINsvHMIDisplay							: REAL;
	rStnExternalTempHALMAXsvHMIDisplay							: REAL;
	
	rStnExternalTempHYSMINsvHMIDisplay							: REAL;
	rStnExternalTempHYSMAXsvHMIDisplay							: REAL;
	
	rStnExternalTempRDYMINsvHMIDisplay							: REAL;
	rStnExternalTempRDYMAXsvHMIDisplay							: REAL;
	
	rStnExternalTemp1stLimitMINsvHMIDisplay						: REAL;
	rStnExternalTemp1stLimitMAXsvHMIDisplay						: REAL;
	
	iStnExternalPreparationTempMINsvHMIDisplay					: INT;
	iStnExternalPreparationTempMAXsvHMIDisplay					: INT;

(* xxxxxxxxxxxxxxxxxxxxxxxxxxxxxxxx Multi Arm Auto Origin Cltr xxxxxxxxxxxxxxxxxxxxxxxxxxxxxxxx*)
(*========================================================================*)

	bAutoOriginStep1: BOOL;
	bAutoOriginStep2: BOOL;
	bAutoOriginStep3: BOOL;
	bAutoOriginStep4: BOOL;
	bAutoOriginStep5: BOOL;
	bAutoOriginStep6: BOOL;
	bAutoOriginStep7: BOOL;
	bAutoOriginStep8: BOOL;
	bAutoOriginStep9: BOOL;

	bMultiArmAutoOriginComplete: BOOL;

(* xxxxxxxxxxxxxxxxxxxxxxxxxxxxxxxx Multi Arm Pnp Cltr xxxxxxxxxxxxxxxxxxxxxxxxxxxxxxxx*)
(*========================================================================*)

	bAllMultiArmBtmPos: BOOL;
	bAllMultiArmTopPos: BOOL;

	bOverallProcessTimeStart: BOOL;
	bOverallProcessTimeReset: BOOL;

	bOverallProcessTimeComplete: BOOL;

	bMultiArmPnpStep1: BOOL;
	bMultiArmPnpStep2: BOOL;
	bMultiArmPnpStep3: BOOL;
	bMultiArmPnpStep4: BOOL;
	bMultiArmPnpStep5: BOOL;
	bMultiArmPnpStep6: BOOL;
	bMultiArmPnpStep7: BOOL;
	bMultiArmPnpStep8: BOOL;
	bMultiArmPnpStep9: BOOL;

(* xxxxxxxxxxxxxxxxxxxxxxxxxxxxxxxx Stn1-3 Station Agitation Process Cltr xxxxxxxxxxxxxxxxxxxxxxxxxxxxxxxx*)
(*========================================================================*)

	bMultiArm1AgiEn: BOOL;
	bMultiArm1AgiInProcess: BOOL;

	bMultiArm2AgiEn: BOOL;
	bMultiArm2AgiInProcess: BOOL;

	bMultiArm3AgiEn: BOOL;
	bMultiArm3AgiInProcess: BOOL;

(* xxxxxxxxxxxxxxxxxxxxxxxxxxxxxxxx Stn1-3 Station Process Cltr xxxxxxxxxxxxxxxxxxxxxxxxxxxxxxxx*)
(*========================================================================*)

	bRecycleMacChillarNoReadySignal  : BOOL;
	bBasketTransferAvailableAlarmBit	: BOOL;
(*Stn1*)

	NoInt 							: INT;

	iStn1ProcessTimeFeedSV			: INT;
	iStn1ProcessTimeSV				: INT;
	iStn1ProcessTimeFeedEV			: INT;

	iStn1SubSeq1					: INT;
	iStn1SubSeq2					: INT;
	iStn1SubSeq3					: INT;
	iStn1SubSeq4					: INT;
	iStn1SubSeq5					: INT;
	iStn1SubSeq6					: INT;
	iStn1SubSeq7					: INT;
	iStn1SubSeq8					: INT;
	iStn1SubSeq9					: INT;
	iStn1SubSeq10					: INT;

	iStn1SubSeq1PV					: INT;
	iStn1SubSeq2PV					: INT;
	iStn1SubSeq3PV					: INT;
	iStn1SubSeq4PV					: INT;
	iStn1SubSeq5PV					: INT;
	iStn1SubSeq6PV					: INT;
	iStn1SubSeq7PV					: INT;
	iStn1SubSeq8PV					: INT;
	iStn1SubSeq9PV					: INT;
	iStn1SubSeq10PV					: INT;

	iMain_Prog_No					: INT;

	iSubProg_No1					: INT;
	iStn1SubProg_no					: INT;

	iStn1RecipeNo					: INT;
	iLdRecipeNo						: INT;
END_VAR

// ---- GVLs/Special_Ctrl/Global_Variables_Special_Persistent.TcGVL
{attribute 'Tc2GvlVarNames'}
VAR_GLOBAL PERSISTENT

(* xxxxxxxxxxxxxxxxxxxxxxxxxxxxxxxx Temperature Cltr xxxxxxxxxxxxxxxxxxxxxxxxxxxxxxxx*)
(*========================================================================*)

	ARfbStnWaterJacketTempControl								: ARRAY [1..iStnQty] OF fbV2_TempControl;
	ARfbStnSubTankTempControl									: ARRAY [1..iStnQty] OF fbV2_TempControl;
	fbJRSInlineHeaterTempControl								: fbV2_TempControl;
	fbIncTempControl											: fbV2_TempControl;
	fbOilSeparatorTempControl									: fbV2_TempControl;


	ARfbStnIncVaporPurgeTempControl								: ARRAY [1..iStnQty] OF fbRawRatioConversionReal;

	ARrStnWaterJacketAnalogInputFineTuneRatio					: ARRAY [1..iStnQty] OF REAL;

	ARrStnWaterJacketTempHYSsv									: ARRAY [1..iStnQty] OF REAL;
	ARrStnWaterJacketTempHALsv									: ARRAY [1..iStnQty] OF REAL;
	ARrStnWaterJacketTempSV										: ARRAY [1..iStnQty] OF REAL;
	ARrStnWaterJacketTempRDYsv									: ARRAY [1..iStnQty] OF REAL;
	ARrStnWaterJacketTemp1stLimitSv								: ARRAY [1..iStnQty] OF REAL;
	ARrStnWaterJacketTemp2ndLimitSv								: ARRAY [1..iStnQty] OF REAL;
	ARiStnWaterJacketPreparationTempSv							: ARRAY [1..iStnQty] OF INT;

	ARrStnSubTankAnalogInputFineTuneRatio						: ARRAY [1..iStnQty] OF REAL;

	ARrStnSubTankTempHYSsv									: ARRAY [1..iStnQty] OF REAL;
	ARrStnSubTankTempHALsv									: ARRAY [1..iStnQty] OF REAL;
	ARrStnSubTankTempSV										: ARRAY [1..iStnQty] OF REAL;
	ARrStnSubTankTempRDYsv									: ARRAY [1..iStnQty] OF REAL;
	ARrStnSubTankTemp1stLimitSv									: ARRAY [1..iStnQty] OF REAL;
	ARrStnSubTankTemp2ndLimitSv								: ARRAY [1..iStnQty] OF REAL;
	ARiStnSubTankPreparationTempSv								: ARRAY [1..iStnQty] OF INT;

	rJRSInlineHeaterAnalogInputFineTuneRatio						: REAL;

	rJRSInlineHeaterTempHYSsv									: REAL;
	rJRSInlineHeaterTempHALsv									: REAL;
	rJRSInlineHeaterTempSV										: REAL;
	rJRSInlineHeaterTempRDYsv									: REAL;
	rJRSInlineHeaterTemp1stLimitSv								: REAL;
	rJRSInlineHeaterTemp2ndLimitSv								: REAL;
	iJRSInlineHeaterPreparationTempSv								: INT;

	rIncAnalogInputFineTuneRatio									: REAL;

	rIncTempHYSsv												: REAL;
	rIncTempHALsv												: REAL;
	rIncTempSV													: REAL;
	rIncTempRDYsv												: REAL;
	rIncTemp1stLimitSv											: REAL;
	rIncTemp2ndLimitSv											: REAL;
	iIncPreparationTempSv										: INT;

	rOilSeparatorTempHYSsv										: REAL;
	rOilSeparatorTempHALsv										: REAL;
	rOilSeparatorTempSV											: REAL;
	rOilSeparatorTempRDYsv										: REAL;
	rOilSeparatorTemp1stLimitSv									: REAL;
	rOilSeparatorTemp2ndLimitSv									: REAL;
	iOilSeparatorPreparationTempSv								: INT;

// 1= Left Top, 2 = Left Bottom, 3= Right Top, 4= Right bottom	
	ARfbStnExternalTempControl									: ARRAY [1..4] OF  fbV2_TempControl;
	ARrStnExternalTempHYSsv										: ARRAY [1..4] OF REAL;
	ARrStnExternalTempHALsv										: ARRAY [1..4] OF REAL;
	ARrStnExternalTempSV										: ARRAY [1..4] OF REAL;
	ARrStnExternalTempRDYsv										: ARRAY [1..4] OF REAL;
	ARrStnExternalTemp1stLimitSv								: ARRAY [1..4] OF REAL;
	ARrStnExternalTemp2ndLimitSv								: ARRAY [1..4] OF REAL;
	ARiStnExternalPreparationTempSv								: ARRAY [1..4] OF INT;

	ARrStnExternalTempHYSMINsv									: ARRAY [1..4] OF REAL;
	ARrStnExternalTempHYSMAXsv									: ARRAY [1..4] OF REAL;
	
	ARrStnExternalTempHALMINsv									: ARRAY [1..4] OF REAL;
	ARrStnExternalTempHALMAXsv									: ARRAY [1..4] OF REAL;
	
	ARrStnExternalTempMINsv										: ARRAY [1..4] OF REAL;
	ARrStnExternalTempMAXsv										: ARRAY [1..4] OF REAL;
	
	ARrStnExternalTempRDYMINsv									: ARRAY [1..4] OF REAL;
	ARrStnExternalTempRDYMAXsv									: ARRAY [1..4] OF REAL;
	
	ARrStnExternalTemp1stLimitMINsv								: ARRAY [1..4] OF REAL;
	ARrStnExternalTemp1stLimitMAXsv								: ARRAY [1..4] OF REAL;
	
	ARiStnExternalPreparationTempMINsv							: ARRAY [1..4] OF INT;
	ARiStnExternalPreparationTempMAXsv							: ARRAY [1..4] OF INT;
(*Agitation Control*)
	DSAgitationParameterStore										: DSPnpAgitationParameter;
	DSAgitationParameter_Pick										: DSPnpAgitationParameter;
	DSAgitationParameter_Transfer									: DSPnpAgitationParameter;
	DSArm2AgitationParameterStore								: DSPnpAgitationParameter;
	DSArm2AgitationParameter_Pick								: DSPnpAgitationParameter;
	DSArm2AgitationParameter_Transfer								: DSPnpAgitationParameter;
(* xxxxxxxxxxxxxxxxxxxxx Multiple Arm Actuator Valve Holding Cltr xxxxxxxxxxxxxxxxxxxxx*)
(*========================================================================*)

	bMultiArm1CylinderUpHolding									: BOOL;
	bMultiArm1CylinderDownHolding								: BOOL;

	bMultiArm2CylinderUpHolding									: BOOL;
	bMultiArm2CylinderDownHolding								: BOOL;

	bMultiArm3CylinderUpHolding									: BOOL;
	bMultiArm3CylinderDownHolding								: BOOL;

	bMultiArm4CylinderUpHolding									: BOOL;
	bMultiArm4CylinderDownHolding								: BOOL;

	bLoadingCylinderUpHolding									: BOOL;
	bLoadingCylinderDownHolding									: BOOL;

	bMultiArmCylinderLeftHolding									: BOOL;
	bMultiArmCylinderRightHolding									: BOOL;

	bMultiArmCylinderClampHolding									: BOOL;
	bMultiArmCylinderUnclampHolding								: BOOL;

(* xxxxxxxxxxxxxxxxxxxxx Multiple Arm Basket Memory Cltr xxxxxxxxxxxxxxxxxxxxx*)
(*========================================================================*)

	bLoadingConvBasketCFM										: BOOL;
	bLoadingConvBasketTRF										: BOOL;

	bLoadingBasketCFM											: BOOL;
	bLoadingBasketTRF											: BOOL;

	bStn1BasketCFM												: BOOL;
	bStn1BasketTRF												: BOOL;

	bStn2BasketCFM												: BOOL;
	bStn2BasketTRF												: BOOL;

	bStn3BasketCFM												: BOOL;
	bStn3BasketTRF												: BOOL;

	bStnbefore4BasketCFM										: BOOL;
	bStnbefore4BasketTRF										: BOOL;

	ARbMultiArmPnpStepHR										: ARRAY[1..10] OF BOOL;
	ARbMultiAutoOriStepHR										: ARRAY[1..10] OF BOOL;

	iLoadingDelayOnSv											: INT;
	iUldStopper2DownTimeDelay									: INT;
	diLdConvDelayTimer											: DINT;

END_VAR

// ---- GVLs/TimeOptimize_Ctrl/Global_Variables_TimeOptimize.TcGVL
{attribute 'Tc2GvlVarNames'}
VAR_GLOBAL PERSISTENT
(*VAR_GLOBAL*)

	bTimeOptimizeDisable								: BOOL;

	ARiCalledTotalProcessTimeStn1					: ARRAY[1..5] OF INT;
	ARiCalledTotalProcessTimeStn2					: ARRAY[1..5] OF INT;
	ARiCalledTotalProcessTimeStn3					: ARRAY[1..5] OF INT;
	ARiCalledTotalProcessTimeStn4					: ARRAY[1..5] OF INT;
	ARiCalledTotalProcessTimeStn5					: ARRAY[1..5] OF INT;
	ARiCalledTotalProcessTimeStn6					: ARRAY[1..5] OF INT;
	ARiCalledTotalProcessTimeStn7					: ARRAY[1..5] OF INT;
	ARiCalledTotalProcessTimeStn8					: ARRAY[1..5] OF INT;
	ARiCalledTotalProcessTimeStn9					: ARRAY[1..5] OF INT;
	ARiCalledTotalProcessTimeStn10					: ARRAY[1..5] OF INT;

(*[][][][][][][][][][][][][][][][][][][][]---fbMasterTimeBlockG2---[][][][][][][][][][][][][][][][][][][][]*)
(*
	fbV2MasterTimeBlockG2_Auto						: fbV2_MasterTimeBlockG2;
*)
(*Input*)
	bMTBStartEN 									: BOOL;
	bMTBScanEN									: BOOL;                         (*bScanOnFlag*)
	bMTBWriteEN 									: BOOL;
	bMTBResetEN 									: BOOL;

(*Output*)
	bMTBScanCompletedFlag							: BOOL;
	bMTBWriteDoneFlag 								: BOOL;
	bMTBResetDoneFlag 								: BOOL;
	bMTBWriteArmDataError 							: BOOL;
	bMTBWriteStnDataError							: BOOL;
	bMTBWriteUldDataError							: BOOL;
	bMTBNoAvailableSlotError 							: BOOL;
	bMTBArmIDAndStnIDAndUldIDNotFound			 	: BOOL;

	bMTBWriteDisable								: BOOL;
	bMTBWriteRetry									: BOOL;
	bMTBWriteExecuteError							: BOOL;

	iMTBNextTransferScanCounter						: INT;
	iMTBNextNotAvailableScanCounter					: INT;
	iMTBNextTransferTime							: INT;
	iMTBNextNotAvailableTime						: INT;

(*[][][][][][][][][][][][][][][][][][][][]---fbTimeBlockSimulatorG2---[][][][][][][][][][][][][][][][][][][][]*)

	fbV2TimeBlockSimulatorG2_Main					: fbV2_TimeBlockSimulatorG2;

(*Input*)
	bSimulateTSEN									: BOOL;

(*Output*)
	bSimulateCompletedFlag							: BOOL;
	iSimulatePercentage								: INT;
	bSimNoSpaceForArmDataToFill					: BOOL;
	bSimNoSpaceForStnDataToFill						: BOOL;
	bSimArmIDAndStnIDNotFound						: BOOL;

	iSimulatedBasketQty								: INT;
	iSimMasterTotalTime								: INT;
	iSimAvarageTimeSec								: INT;

	rSimBasketQtyPerHour								: REAL;

(*[][][][][][][][][][][][][][][][][][][][]---fbFBPTimeTrackerG2---[][][][][][][][][][][][][][][][][][][][]*)

	DSTimeTrackerInput								: DSV2_TimeTrackerInput;

(*Input*)
	bTrackerStartEN									: BOOL;

	iCallRecipeTimeBlock_ProductRecipeNo 			: INT;

	iSimulatorProductRecipeNo							: INT;
	iUserDefineProductRecipeNo						: INT;
	iTrackerProductRecipeNo 							: INT;
	iDisplayUserDefineProductRecipeNo				:INT;

(*Output*)

	bTrackerCompleted 								: BOOL;
	bNoUldStnIDErr									: BOOL;
	bInvalidCallRecipeTimeBlockNo					: BOOL;
	bCallRTB_NoTrackerInfo							: BOOL;
	bCallRTB_CallOK 									: BOOL;
	bCallModeError									: BOOL;


(*[][][][][][][][][][][][][][][][][][][][]---fbMasterTimeBlockG2---[][][][][][][][][][][][][][][][][][][][]*)

(*Input*)
	iMTBScanCompleteDelayOnTime_ms				: INT := 1000;
	iMTBWriteRetryQty								: INT := 3;
	iMTBWriteRetryDelayTimeSec						: INT := 2;

	AR3SiMasterTimeBlockArm_MTB		 			: ARRAY[1..iArmQty, 1..iMasterBlockQty, 1..3] OF INT;
	AR3SiMasterTimeBlockStn_MTB					: ARRAY[1..iStnQty, 1..iMasterBlockQty, 1..3] OF INT;
	AR3SiMasterTimeBlockUld_MTB					: ARRAY[1..iUldStnQty, 1..iMasterBlockQty, 1..3] OF INT;

(*Output*)
	ARbMTBArmProgress								: ARRAY [1..iArmQty] OF BOOL;

(*[][][][][][][][][][][][][][][][][][][][]---fbTimeBlockSimulatorG2---[][][][][][][][][][][][][][][][][][][][]*)

(*Input*)
	AR3SiMasterTimeBlockArm_Simulator 				: ARRAY[1..iArmQty, 1..iMasterBlockQty, 1..9] OF INT;
	AR3SiMasterTimeBlockStn_Simulator				: ARRAY[1..iStnQty, 1..iMasterBlockQty, 1..9] OF INT;

(*Output*)
	ARiSimBasketTimeStamp 							: ARRAY [1..100] OF INT;


(*[][][][][][][][][][][][][][][][][][][][]---fbFBPTimeTrackerG2---[][][][][][][][][][][][][][][][][][][][]*)

	fbV2FBPTimeTrackerG3_Main						: fbV2_FBPTimeTrackerG3;


(*Input*)

	bTrackerReset 									: ARRAY [0..iProductRecipeArrayQty] OF BOOL;

	ARbReset 										: ARRAY [0..iProductRecipeArrayQty] OF BOOL;
	ARbArmSt 										: ARRAY [1..iArmQty] OF BOOL; (*Activated Bit*)
	iCountFilterTime_Sec 								: INT := 2;
	AR2SiBufferRecipeTimeBlock 						: ARRAY[1..iRecipeBlockQty, 1..9] OF INT;

	ARbBusyLinkUpStnEn 								: ARRAY [1..iBusyLinkUpSetQty] OF BOOL;
	AR2siStnBusyLinkUpStn 							: ARRAY [1..iBusyLinkUpSetQty, 1..iBusyLinkUpStnQty] OF INT;


(*Output*)

	AR2SiCalledRecipeTimeBlockNoCallArmTime 		: ARRAY[1..iRecipeBlockQty, 1..9] OF INT;
	AR2SiCalledRecipeTimeBlockWithCallArmTime 		: ARRAY[1..iRecipeBlockQty, 1..9] OF INT;

	ARbProductRecipeTimeBlockAvailable				: ARRAY [0..iProductRecipeArrayQty] OF BOOL;

	AR2SiArmRunningTime							: ARRAY [1..iRecipeBlockQty, 1..iArmQty] OF INT;
	ARiStnRunningTime								: ARRAY [1..iRecipeBlockQty] OF INT;

(*[][][][][][][][][][][][][][][][][][][][]---Multiple FB Used---[][][][][][][][][][][][][][][][][][][][]*)

(*	AR2SiRecipeTimeBlock							: ARRAY [1..iRecipeBlockQty, 1..3] OF INT;
	ARbSkipStation									: ARRAY [1..iStnQty] OF BOOL;

	ARiZoneAddress									: ARRAY [1..iRecipeBlockQty] OF INT;
	ARiZoneArea										: ARRAY [1..iRecipeBlockQty] OF INT;
*)	ARiArmID										: ARRAY [1..iArmQty] OF INT;


(*[][][][][][][][][][][][][][][][][][][][]---fbFBPTimeTrackerG2---[][][][][][][][][][][][][][][][][][][][]*)


(*Input*)
	ARbAlternateStnEn 								: ARRAY [1..iAlternateSetQty] OF BOOL;
	AR2siAlternateStn 									: ARRAY [1..iAlternateSetQty, 1..iAlternateStnQty] OF INT;

END_VAR

// ---- GVLs/UserCtrl/GVL_UserCtrl.TcGVL

VAR_GLOBAL
	
// HMI CONTROL

	bUserNameLoginPageOn	: BOOL;
	bUserNameEditPageOn	: BOOL;
	bPageConfirmPageOn: BOOL;
//		

	bAutoModeLock : BOOL;

	userpassword:ARRAY [1..5] OF STRING;
	username:ARRAY [1..5] OF WSTRING;
	sUserGroupName:ARRAY [1..5] OF WSTRING;
	userlogin : ARRAY [1..5] OF BOOL;
		
	sActiveUserGroupname: WSTRING;
	
	bUserGroupPageON: BOOL;
	bUserPageCreateON :BOOL;
	bUserPageEditON	: BOOL;
	iCurrentUserGroupID :INT;
	sCurrentPwField: STRING;
	sNewPwField: STRING;
	sConfirmPwField: STRING;
	sPwField: STRING;
		
	// LKT Test
	
	fbHmiTF1800_UserlevelManagement : FB3_HmiTF1800_UserlevelManagement;
	
		//For F HmiTF1800
		
			// Input
			bLoginPB 					: BOOL;
			bLogoutPB 					: BOOL;
			iLoginNameId 				: INT; // The LoginName selection in HMI during User Login Pop-up Screen, the choosen user will translated as Array ID No and pass here.
			sPasswordField 				: STRING; // Similar to Var In/Out so that i can clear the password if login failed
			
			iUM_SelectedLoginNameId	 	: INT;		// User Management - Selected Login Name ID (Array No)
		
			sUM_CurrentPassword			: STRING;	// User Management - Current Password (For password change only)
			sUM_NewPassword				: STRING;	// User Management - New Password (For password change or new user registration)
			sUM_ConfirmPassword			: STRING;	// User Management - New Password (For password change or new user registration)
		
			sUM_NewUserLoginName		: STRING;	// User Management - New User Login Name
			sUM_NewUserGroupId			: INT;		// User Management - Select from UserGroupList
		
			sUM_NewUserOperatorIdentifier	: STRING;
			sUM_NewUserActorType			: eActor;
			sUM_NewUserLastName				: STRING;
			sUM_NewUserFirstName			: STRING;
			
			bUM_CreatePB				: BOOL;		// User Management - Button for New User creation
			bUM_EditPB					: BOOL;		// User Management - Button for Edit User
			bUM_DeletePB				: BOOL;		// User Management - Button for Delete User
			bUM_EnablePB				: BOOL; 	// to Enable selected User
			bUM_DisablePB				: BOOL; 	// to Temporary Disable selected User
			bUM_ConfirmPB				: BOOL;		// for Edit, Delete and Disable used. click to save
			bUM_ReturnPB				: BOOL;		// for Edit, Delete and Disable used, click to return without save.
			
			//Output
			dsHmiUserStatus_Active		: DS_HmiUserStatus;
			dsHmiUserStatus_Login		: DS_HmiUserStatus;
			dsHmiUserStatus_Logout		: DS_HmiUserStatus;
			
			wsActiveUserGroupName		: WSTRING;
			sMessage					: STRING;

			

END_VAR

// ---- GVLs/XML_Ctrl/XML.TcGVL
{attribute 'Tc2GvlVarNames'}
VAR_GLOBAL

	XML_ImportExport 										: ARRAY [1..iProductRecipeArrayQty] OF DS_XML_InputOutput;

	sFilePath				:T_MaxString;


	bRead					: BOOL;

	FBXmlSrvRead1			:  FB_XmlSrvRead;
	ePath 					: E_OpenPath := PATH_GENERIC;
	nMode 					: WORD := XMLSRV_ADDMISSING;
(*	sFilePath1				:T_MaxString:='C:\Users\SFQ\Desktop\File1.xml';*)
	sXPath					:T_MaxString:='/dataentry/MAIN.value1';
	bEXERead1				: BOOL;


	bEXEWrite1				: BOOL;
	FBXmlSrvWrite1			:  FB_XmlSrvWrite;





	Filename: STRING;
	string1: STRING;
	string2: STRING;
	step: INT;
	bImport: BOOL;
	bExport: BOOL;
	bWriteDone				: BOOL;
	bReadDone				: BOOL;



	iFLStnNo: INT;
	iFLRcpNo: INT;
	iRcpNo: INT;

	bImport_file: BOOL;
	bExport_file: BOOL;
	bImportDone: BOOL;
	iFLStnNo1: INT;
	iFLStnNo2: INT;
	bExportDone: BOOL;



	fbV3XML_Handler_Server					: fbV3_XML_Handler;
	bErrorRst_Server							: BOOL;
	bXMLServerBusyFlag						: BOOL;
	bXMLServerErrorFlag						: BOOL;
	udXMLServerErrorID						: UDINT;

	fbV3XML_Handler_Local					: fbV3_XML_Handler;
	bErrorRst_Local							: BOOL;
	bXMLLocalBusyFlag						: BOOL;
	bXMLLocalErrorFlag						: BOOL;
	udXMLLocalErrorID						: UDINT;


	iLocalImportHS							: INT;
	iLocalExportHS							: INT;
	iLocalDeleteAllHS							: INT;
	iLocalImportExportRecipeNo				: INT;


END_VAR

// ---- POUs/MAIN.TcPOU
PROGRAM MAIN
VAR
		tPowerOnDelayOn: TON;
		tPowerOnDelayOff: TON;
dummy: BOOL;
END_VAR

// NodeRed_BasketLog(); 

// ARwActualMapDI[2].6;
ArbDI[eX10106_GeneralPhaseSequenceRelayMcb_Trip];
Bootup_Shutdown_ctrl();
XML_PersistentCtrl();
//UpsSignal();
//PID_Ctrl_Test(); //LKT Basic PID
SerialCom();

//IF bMainCtrl THEN

OPC_UA_MAP();
	
Modbus_test();
Manual_ImportExport_Others();

Barcode_Reg();
	
Internal_Mapping();
IO_Mapping();

(*zAutoMode*)
(*============================*)
AutoMain();
AutoMain_AddON();
AutoOriginCtrl();
AutoPreparationCtrl();
AutoPreparationCtrl_ST();
AutoStartCtrl();
HMI_Page_Control();

(*A_StandardStructureProgram*)
(*============================*)

stClockPulseBlink();
stGetCurrentTime();
stUPSStatusMonitoring();
stWritePersistentData();

(*Aa_HmiVariableCtrl*)
(*============================*)
HMIValueKeyInCtrl();

(*AgitationMechanismCtrl*)
(*============================*)
AgitationMechanismCtrl();

